(* CODESYS project MC516.project
   CompiledLibraryCompatibilityVersion: LeadSysStudio V3.5 SP15 Patch 4
   Title: MC516

Project tree, tasks and I/O mapping:
  Device : MC516, Leadshine Technology Co., Ltd., order no. 516101, version 3.5.15.40
      settings: RetainMode = 0; RetainStartAddr = 20480; RetainEndAddr = 524288; RetainSize = 524288
    application Application
      libraries: Standard, * (System)
      task EtherCAT_Master_Leadshine_A (cyclic, interval 2000 µs, priority 0) calls EtherCAT_Master_Leadshine_A.EtherCAT_Task, M
      program M [ST]: io, motion, save_check, save_apply, work
      DataMain/
        data type HMIData
        data type SaveData
      function block AxisFB [ST]: calculate_home_delta_μ, follow
      Enum/
        data type State
        data type JogType
      Object/
        data type Button
        data type Cylinder
        data type AxisEC
        data type AxisECFollow
        data type Problem
      function StateNext [ST]
      DataWork/
        data type SupplyData
        data type WorkData
        data type CutData
      function block CutFB [ST]
      visualisation Visualization
      function block SupplyFB [ST]
      Symbols
      global variables PersistentVars
      function block AxisFBSetTorqueLimit [ST]
      function block SimpleMotion [ST]
    Resource Usage
    Device Diagnose
    Network Configuration
      LocalBus Config
    SoftMotion General Axis Pool
      JogEncoder : SMC_FreeEncoder, 3S - Smart Software Solutions GmbH, order no. 1805, version 3.5.5.0
          settings: wDriveID = 3; dwRatioTechUnitsDenom = 400; ScalingIncs = 400
    High_Speed_IO_Module : High Speed IO, Leadshine Technology Co., Ltd., version 3.5.15.40
        settings: HS_IO_Mode_0.High In IO Mode 0 = 196611; HS_IO_Mode_0.High In IO Mode 2 = 196611; Counter_Mask = 5; Ioin_Mask = 19; HS counter 1.Counter_CountMode = 1; HS counter 2.Counter_CountMode = 1; HS counter 3.Counter_SetWorkMode = 2; HS counter 3.Counter_CountMode = 1; InputFilter Para.Time_In0 = 2; InputFilter Para.Time_In1 = 2; InputFilter Para.Time_In4 = 2
        unmapped channels: Genral_IO_IN, Genral_IO_Out
    LocalBus_Master_Module : LocalBus Master, Leadshine Technology Co., Ltd., version 3.5.15.40
    EtherCAT_Master_Leadshine_A : EtherCAT Master SoftMotion, 3S - Smart Software Solutions GmbH, version 3.5.16.30
        settings: MasterCycleTime = 2000; NetworkName = 'ecat'; SelectNetworkByName = TRUE; SrcAddress1 = 10; SrcAddress2 = 889192738
      XINJE_DS5C1_CoE_Drive_Rev4_0 : XINJE-DS5C1 EtherCAT(CoE) Drive Rev4.0 v3.7.70, Xinje Electronics, Inc., order no. XINJE-DS5C1 CoE Drive Rev4.0, version Revision=16#20201207
          settings: Number of Inputs = 6; Number of Infos about Inputs = 6; StationAlias = 1; Sync.Length = 17; FMMU.Length = 17; DC sync0 cycletime = 2000; DC sync1 cycletime = 2000; Number of SDO = 6; Interpolation time period.Value = 2; RxTxPdo.NumberofEntries = 6; RxTxPdo.Index = 16#1A00; RxTxPdo.DependOnSlot = False; RxTxPdo.DependOnSlotGroup = False; RxTxPdo.OverwrittenByModule = False; Status Word.Offset = 0; Status Word.DependOnSlot = False; Status Word.DependOnSlotGroup = False; ActualPosition.Offset = 0; ActualPosition.DependOnSlot = False; ActualPosition.DependOnSlotGroup = False; Velocity actual value.Offset = 0; Velocity actual value.DependOnSlot = False; Velocity actual value.DependOnSlotGroup = False; ActualTorque.Offset = 0; ActualTorque.DependOnSlot = False; ActualTorque.DependOnSlotGroup = False; ModeOfOperationDisplay.Offset = 0; ModeOfOperationDisplay.DependOnSlot = False; ModeOfOperationDisplay.DependOnSlotGroup = False; Index = 16#5000; SubIndex = 0; Size = 32; Offset = 0; DependOnSlot = False; DependOnSlotGroup = False; Status Word.Default = ''; Status Word.Comment = ''; ActualPosition.Default = ''; ActualPosition.Comment = ''; Velocity actual value.Default = '';
            Velocity actual value.Comment = ''; ActualTorque.Default = ''; ActualTorque.Comment = ''; ModeOfOperationDisplay.Default = ''; ModeOfOperationDisplay.Comment = ''; Name = 'Encode Single Position'; DataType = 'DINT'; Default = ''; Comment = ''
          unmapped channels: Control Word, TargetPosition, TargetVelocity, TargetTorque, ModeOfOperation, Status Word, ActualPosition, Velocity actual value, ActualTorque, ModeOfOperationDisplay, Encode Single Position
        Axis : Axis, 3S - Smart Software Solutions GmbH, order no. 0, version 4.6.1.0
            settings: wDriveID = 0; dwRatioTechUnitsDenom = 1; eRampType = 3; Number of pulses for one revolution = 131072; The displacement for one revolution of the workbench = 131072; Gear ratio molecule = 1; Gear ratio denominator = 1; ScalingIncs = 131072; InvertDirection = False; AdrOffset_8010 = 4; BitOffset_8010 = 0; BitLength_8010 = 16; Address_8010 = '%QW2'; Type_8010 = 'UINT'; AddressPointer_8010 = ADR(%QW2); AdrOffset_8020 = 8; BitOffset_8020 = 0; BitLength_8020 = 32; Address_8020 = '%QD2'; Type_8020 = 'DINT'; AddressPointer_8020 = ADR(%QD2); AdrOffset_8030 = 12; BitOffset_8030 = 0; BitLength_8030 = 32; Address_8030 = '%QD3'; Type_8030 = 'DINT'; AddressPointer_8030 = ADR(%QD3); AdrOffset_8040 = 16; BitOffset_8040 = 0; BitLength_8040 = 16; Address_8040 = '%QW8'; Type_8040 = 'INT'; AddressPointer_8040 = ADR(%QW8); AdrOffset_8050 = 18; BitOffset_8050 = 0; BitLength_8050 = 8; Address_8050 = '%QB18'; Type_8050 = 'SINT'; AddressPointer_8050 = ADR(%QB18); AdrOffset_8060 = 4294967295;
              BitOffset_8060 = 0; BitLength_8060 = 0; Address_8060 = ''; Type_8060 = ''; AddressPointer_8060 = 0; AdrOffset_8070 = 4294967295; BitOffset_8070 = 0; BitLength_8070 = 0; Address_8070 = ''; Type_8070 = ''; AddressPointer_8070 = 0; AdrOffset_8080 = 4294967295; BitOffset_8080 = 0; BitLength_8080 = 0; Address_8080 = ''; Type_8080 = ''; AddressPointer_8080 = 0; AdrOffset_8090 = 4294967295; BitOffset_8090 = 0; BitLength_8090 = 0; Address_8090 = ''; Type_8090 = ''; AddressPointer_8090 = 0; AdrOffset_8510 = 4; BitOffset_8510 = 0; BitLength_8510 = 16; Address_8510 = '%IW2'; Type_8510 = 'UINT'; AddressPointer_8510 = ADR(%IW2); AdrOffset_8520 = 8; BitOffset_8520 = 0; BitLength_8520 = 32; Address_8520 = '%ID2'; Type_8520 = 'DINT'; AddressPointer_8520 = ADR(%ID2); AdrOffset_8530 = 12; BitOffset_8530 = 0; BitLength_8530 = 32; Address_8530 = '%ID3'; Type_8530 = 'DINT';
              AddressPointer_8530 = ADR(%ID3); AdrOffset_8540 = 16; BitOffset_8540 = 0; BitLength_8540 = 16; Address_8540 = '%IW8'; Type_8540 = 'INT'; AddressPointer_8540 = ADR(%IW8); AdrOffset_8550 = 18; BitOffset_8550 = 0; BitLength_8550 = 8; Address_8550 = '%IB18'; Type_8550 = 'SINT'; AddressPointer_8550 = ADR(%IB18); AdrOffset_8560 = 4294967295; BitOffset_8560 = 0; BitLength_8560 = 0; Address_8560 = ''; Type_8560 = ''; AddressPointer_8560 = 0; AdrOffset_8570 = 4294967295; BitOffset_8570 = 0; BitLength_8570 = 0; Address_8570 = ''; Type_8570 = ''; AddressPointer_8570 = 0; AdrOffset_8580 = 4294967295; BitOffset_8580 = 0; BitLength_8580 = 0; Address_8580 = ''; Type_8580 = ''; AddressPointer_8580 = 0; AdrOffset_8590 = 4294967295; BitOffset_8590 = 0; BitLength_8590 = 0; Address_8590 = ''; Type_8590 = ''; AddressPointer_8590 = 0; AdrOffset_8600 = 4294967295; BitOffset_8600 = 0; BitLength_8600 = 0;
              Address_8600 = ''; Type_8600 = ''; AddressPointer_8600 = 0; AdrOffset_8600 = 4294967295; BitOffset_8600 = 0; BitLength_8600 = 0; Address_8610 = ''; Type_8610 = ''; AddressPointer_8610 = 0; AdrOffset_8620 = 4294967295; BitOffset_8620 = 0; BitLength_8620 = 0; Address_8620 = ''; Type_8620 = ''; AddressPointer_8620 = 0
      XINJE_DS5C1_CoE_Drive_Rev4_0_1 : XINJE-DS5C1 EtherCAT(CoE) Drive Rev4.0 v3.7.70, Xinje Electronics, Inc., order no. XINJE-DS5C1 CoE Drive Rev4.0, version Revision=16#20201207
          settings: Number of Inputs = 6; Number of Infos about Inputs = 6; StationAlias = 1; Optional = False; DeviceIdenticationADO = 0; DeviceIdenticationMode = 0; Sync.Length = 17; FMMU.Length = 17; DC sync0 cycletime = 2000; DC sync1 cycletime = 2000; Number of SDO = 5; Interpolation time period.Value = 2; RxTxPdo.NumberofEntries = 6; RxTxPdo.Index = 16#1A00; RxTxPdo.DependOnSlot = False; RxTxPdo.DependOnSlotGroup = False; RxTxPdo.OverwrittenByModule = False; Status Word.Offset = 0; Status Word.DependOnSlot = False; Status Word.DependOnSlotGroup = False; ActualPosition.Offset = 0; ActualPosition.DependOnSlot = False; ActualPosition.DependOnSlotGroup = False; Velocity actual value.Offset = 0; Velocity actual value.DependOnSlot = False; Velocity actual value.DependOnSlotGroup = False; ActualTorque.Offset = 0; ActualTorque.DependOnSlot = False; ActualTorque.DependOnSlotGroup = False; ModeOfOperationDisplay.Offset = 0; ModeOfOperationDisplay.DependOnSlot = False; ModeOfOperationDisplay.DependOnSlotGroup = False; Index = 16#5000; SubIndex = 0; Size = 32; Offset = 0; DependOnSlot = False; DependOnSlotGroup = False; Status Word.Default = ''; Status Word.Comment = '';
            ActualPosition.Default = ''; ActualPosition.Comment = ''; Velocity actual value.Default = ''; Velocity actual value.Comment = ''; ActualTorque.Default = ''; ActualTorque.Comment = ''; ModeOfOperationDisplay.Default = ''; ModeOfOperationDisplay.Comment = ''; Name = 'Encode Single Position'; DataType = 'DINT'; Default = ''; Comment = ''
          unmapped channels: Control Word, TargetPosition, TargetVelocity, TargetTorque, ModeOfOperation, Status Word, ActualPosition, Velocity actual value, ActualTorque, ModeOfOperationDisplay, Encode Single Position
        Axis_1 : Axis, 3S - Smart Software Solutions GmbH, order no. 0, version 4.6.1.0
            settings: dwRatioTechUnitsDenom = 1; eRampType = 3; Number of pulses for one revolution = 131072; The displacement for one revolution of the workbench = 131072; Gear ratio molecule = 1; Gear ratio denominator = 1; ScalingIncs = 131072; InvertDirection = False; AdrOffset_8010 = 20; BitOffset_8010 = 0; BitLength_8010 = 16; Address_8010 = '%QW10'; Type_8010 = 'UINT'; AddressPointer_8010 = ADR(%QW10); AdrOffset_8020 = 24; BitOffset_8020 = 0; BitLength_8020 = 32; Address_8020 = '%QD6'; Type_8020 = 'DINT'; AddressPointer_8020 = ADR(%QD6); AdrOffset_8030 = 28; BitOffset_8030 = 0; BitLength_8030 = 32; Address_8030 = '%QD7'; Type_8030 = 'DINT'; AddressPointer_8030 = ADR(%QD7); AdrOffset_8040 = 32; BitOffset_8040 = 0; BitLength_8040 = 16; Address_8040 = '%QW16'; Type_8040 = 'INT'; AddressPointer_8040 = ADR(%QW16); AdrOffset_8050 = 34; BitOffset_8050 = 0; BitLength_8050 = 8; Address_8050 = '%QB34'; Type_8050 = 'SINT'; AddressPointer_8050 = ADR(%QB34); AdrOffset_8060 = 4294967295; BitOffset_8060 = 0;
              BitLength_8060 = 0; Address_8060 = ''; Type_8060 = ''; AddressPointer_8060 = 0; AdrOffset_8070 = 4294967295; BitOffset_8070 = 0; BitLength_8070 = 0; Address_8070 = ''; Type_8070 = ''; AddressPointer_8070 = 0; AdrOffset_8080 = 4294967295; BitOffset_8080 = 0; BitLength_8080 = 0; Address_8080 = ''; Type_8080 = ''; AddressPointer_8080 = 0; AdrOffset_8090 = 4294967295; BitOffset_8090 = 0; BitLength_8090 = 0; Address_8090 = ''; Type_8090 = ''; AddressPointer_8090 = 0; AdrOffset_8510 = 24; BitOffset_8510 = 0; BitLength_8510 = 16; Address_8510 = '%IW12'; Type_8510 = 'UINT'; AddressPointer_8510 = ADR(%IW12); AdrOffset_8520 = 28; BitOffset_8520 = 0; BitLength_8520 = 32; Address_8520 = '%ID7'; Type_8520 = 'DINT'; AddressPointer_8520 = ADR(%ID7); AdrOffset_8530 = 32; BitOffset_8530 = 0; BitLength_8530 = 32; Address_8530 = '%ID8'; Type_8530 = 'DINT'; AddressPointer_8530 = ADR(%ID8);
              AdrOffset_8540 = 36; BitOffset_8540 = 0; BitLength_8540 = 16; Address_8540 = '%IW18'; Type_8540 = 'INT'; AddressPointer_8540 = ADR(%IW18); AdrOffset_8550 = 38; BitOffset_8550 = 0; BitLength_8550 = 8; Address_8550 = '%IB38'; Type_8550 = 'SINT'; AddressPointer_8550 = ADR(%IB38); AdrOffset_8560 = 4294967295; BitOffset_8560 = 0; BitLength_8560 = 0; Address_8560 = ''; Type_8560 = ''; AddressPointer_8560 = 0; AdrOffset_8570 = 4294967295; BitOffset_8570 = 0; BitLength_8570 = 0; Address_8570 = ''; Type_8570 = ''; AddressPointer_8570 = 0; AdrOffset_8580 = 4294967295; BitOffset_8580 = 0; BitLength_8580 = 0; Address_8580 = ''; Type_8580 = ''; AddressPointer_8580 = 0; AdrOffset_8590 = 4294967295; BitOffset_8590 = 0; BitLength_8590 = 0; Address_8590 = ''; Type_8590 = ''; AddressPointer_8590 = 0; AdrOffset_8600 = 4294967295; BitOffset_8600 = 0; BitLength_8600 = 0; Address_8600 = '';
              Type_8600 = ''; AddressPointer_8600 = 0; AdrOffset_8600 = 4294967295; BitOffset_8600 = 0; BitLength_8600 = 0; Address_8610 = ''; Type_8610 = ''; AddressPointer_8610 = 0; AdrOffset_8620 = 4294967295; BitOffset_8620 = 0; BitLength_8620 = 0; Address_8620 = ''; Type_8620 = ''; AddressPointer_8620 = 0
      XINJE_DS5C1_CoE_Drive_Rev4_0_2 : XINJE-DS5C1 EtherCAT(CoE) Drive Rev4.0 v3.7.70, Xinje Electronics, Inc., order no. XINJE-DS5C1 CoE Drive Rev4.0, version Revision=16#20201207
          settings: Number of Inputs = 6; Number of Infos about Inputs = 6; StationAlias = 1; Optional = False; DeviceIdenticationADO = 0; DeviceIdenticationMode = 0; Sync.Length = 17; FMMU.Length = 17; DC sync0 cycletime = 2000; DC sync1 cycletime = 2000; Number of SDO = 8; Interpolation time period.Value = 2; RxTxPdo.NumberofEntries = 6; RxTxPdo.Index = 16#1A00; RxTxPdo.DependOnSlot = False; RxTxPdo.DependOnSlotGroup = False; RxTxPdo.OverwrittenByModule = False; Status Word.Offset = 0; Status Word.DependOnSlot = False; Status Word.DependOnSlotGroup = False; ActualPosition.Offset = 0; ActualPosition.DependOnSlot = False; ActualPosition.DependOnSlotGroup = False; Velocity actual value.Offset = 0; Velocity actual value.DependOnSlot = False; Velocity actual value.DependOnSlotGroup = False; ActualTorque.Offset = 0; ActualTorque.DependOnSlot = False; ActualTorque.DependOnSlotGroup = False; ModeOfOperationDisplay.Offset = 0; ModeOfOperationDisplay.DependOnSlot = False; ModeOfOperationDisplay.DependOnSlotGroup = False; Index = 16#5000; SubIndex = 0; Size = 32; Offset = 0; DependOnSlot = False; DependOnSlotGroup = False; Status Word.Default = ''; Status Word.Comment = '';
            ActualPosition.Default = ''; ActualPosition.Comment = ''; Velocity actual value.Default = ''; Velocity actual value.Comment = ''; ActualTorque.Default = ''; ActualTorque.Comment = ''; ModeOfOperationDisplay.Default = ''; ModeOfOperationDisplay.Comment = ''; Name = 'Encode Single Position'; DataType = 'DINT'; Default = ''; Comment = ''
          unmapped channels: Control Word, TargetPosition, TargetVelocity, TargetTorque, ModeOfOperation, Status Word, ActualPosition, Velocity actual value, ActualTorque, ModeOfOperationDisplay, Encode Single Position
        Axis_2 : Axis, 3S - Smart Software Solutions GmbH, order no. 0, version 4.6.1.0
            settings: wDriveID = 2; dwRatioTechUnitsDenom = 1; iMovementType = 0; fPositionPeriod = 360000; eRampType = 3; Number of pulses for one revolution = 131072; The displacement for one revolution of the workbench = 131072; Gear ratio molecule = 1; Gear ratio denominator = 1; ScalingIncs = 131072; InvertDirection = False; AdrOffset_8010 = 36; BitOffset_8010 = 0; BitLength_8010 = 16; Address_8010 = '%QW18'; Type_8010 = 'UINT'; AddressPointer_8010 = ADR(%QW18); AdrOffset_8020 = 40; BitOffset_8020 = 0; BitLength_8020 = 32; Address_8020 = '%QD10'; Type_8020 = 'DINT'; AddressPointer_8020 = ADR(%QD10); AdrOffset_8030 = 44; BitOffset_8030 = 0; BitLength_8030 = 32; Address_8030 = '%QD11'; Type_8030 = 'DINT'; AddressPointer_8030 = ADR(%QD11); AdrOffset_8040 = 48; BitOffset_8040 = 0; BitLength_8040 = 16; Address_8040 = '%QW24'; Type_8040 = 'INT'; AddressPointer_8040 = ADR(%QW24); AdrOffset_8050 = 50; BitOffset_8050 = 0; BitLength_8050 = 8; Address_8050 = '%QB50'; Type_8050 = 'SINT';
              AddressPointer_8050 = ADR(%QB50); AdrOffset_8060 = 4294967295; BitOffset_8060 = 0; BitLength_8060 = 0; Address_8060 = ''; Type_8060 = ''; AddressPointer_8060 = 0; AdrOffset_8070 = 4294967295; BitOffset_8070 = 0; BitLength_8070 = 0; Address_8070 = ''; Type_8070 = ''; AddressPointer_8070 = 0; AdrOffset_8080 = 4294967295; BitOffset_8080 = 0; BitLength_8080 = 0; Address_8080 = ''; Type_8080 = ''; AddressPointer_8080 = 0; AdrOffset_8090 = 4294967295; BitOffset_8090 = 0; BitLength_8090 = 0; Address_8090 = ''; Type_8090 = ''; AddressPointer_8090 = 0; AdrOffset_8510 = 44; BitOffset_8510 = 0; BitLength_8510 = 16; Address_8510 = '%IW22'; Type_8510 = 'UINT'; AddressPointer_8510 = ADR(%IW22); AdrOffset_8520 = 48; BitOffset_8520 = 0; BitLength_8520 = 32; Address_8520 = '%ID12'; Type_8520 = 'DINT'; AddressPointer_8520 = ADR(%ID12); AdrOffset_8530 = 52; BitOffset_8530 = 0; BitLength_8530 = 32;
              Address_8530 = '%ID13'; Type_8530 = 'DINT'; AddressPointer_8530 = ADR(%ID13); AdrOffset_8540 = 56; BitOffset_8540 = 0; BitLength_8540 = 16; Address_8540 = '%IW28'; Type_8540 = 'INT'; AddressPointer_8540 = ADR(%IW28); AdrOffset_8550 = 58; BitOffset_8550 = 0; BitLength_8550 = 8; Address_8550 = '%IB58'; Type_8550 = 'SINT'; AddressPointer_8550 = ADR(%IB58); AdrOffset_8560 = 4294967295; BitOffset_8560 = 0; BitLength_8560 = 0; Address_8560 = ''; Type_8560 = ''; AddressPointer_8560 = 0; AdrOffset_8570 = 4294967295; BitOffset_8570 = 0; BitLength_8570 = 0; Address_8570 = ''; Type_8570 = ''; AddressPointer_8570 = 0; AdrOffset_8580 = 4294967295; BitOffset_8580 = 0; BitLength_8580 = 0; Address_8580 = ''; Type_8580 = ''; AddressPointer_8580 = 0; AdrOffset_8590 = 4294967295; BitOffset_8590 = 0; BitLength_8590 = 0; Address_8590 = ''; Type_8590 = ''; AddressPointer_8590 = 0; AdrOffset_8600 = 4294967295;
              BitOffset_8600 = 0; BitLength_8600 = 0; Address_8600 = ''; Type_8600 = ''; AddressPointer_8600 = 0; AdrOffset_8600 = 4294967295; BitOffset_8600 = 0; BitLength_8600 = 0; Address_8610 = ''; Type_8610 = ''; AddressPointer_8610 = 0; AdrOffset_8620 = 4294967295; BitOffset_8620 = 0; BitLength_8620 = 0; Address_8620 = ''; Type_8620 = ''; AddressPointer_8620 = 0
  text list GlobalTextList
*)

// Device/Application/DataMain/HMIData
{ attribute 'pack_mode' := ''}
TYPE HMIData :
STRUCT
	//
	sv: SaveData;
	sv_trigger: BOOL;
	sv_need_check: BOOL;
	sv_need: BOOL;
	//
	plc_ready: BOOL;
	hmi_ready: BOOL;
	run: BOOL;
	stop: BOOL;
	home: BOOL;
	problem_fix: ARRAY[0..7] OF BOOL;
	//
	supply_test: BOOL;
	supply_arm_clamp_holder: BOOL;
	supply_arm_clamp: BOOL;
	supply_spindle_clamp: BOOL;
	supply_spindle_extract: BOOL;
	cut_spindle_run: BOOL;
	hydraulic_run: BOOL;
	jog_micro_per_sec_or_rev: UINT;
	//
	view_input: ARRAY[0..15] OF BOOL;
	view_input_jog_index: UINT;
	view_input_jog_micro: DINT;
	view_output: ARRAY[0..15] OF BOOL;
	//
	view_can_run: BOOL;
	view_can_stop: BOOL;
	view_can_home: BOOL;
	view_auto: BOOL;
	view_manual: BOOL;
	//
	view_axis_encoder: ARRAY[0..2] OF DINT;
	view_axis_micro: ARRAY[0..2] OF UDINT;
	view_axis_mNm: ARRAY[0..2] OF UDINT;
	view_cut_spindle_run_ing: BOOL;
	view_cut_spindle_rpm: UDINT;
	//
	view_supply_test: ARRAY[0..4] OF BOOL;
	//
	view_problem: ARRAY[0..7] OF BOOL;
	view_cycle_count: UDINT;
	view_cycle_time_msec: UDINT;
	//
	view_state: ARRAY[0..7] OF INT;
END_STRUCT
END_TYPE

// Device/Application/DataMain/SaveData
{ attribute 'pack_mode' := ''}
TYPE SaveData :
STRUCT
	set_done: BOOL;
	////////
	//SAME//
	////////
	cylinder_n_delay_msec: ARRAY[0..3] OF UINT;
	cylinder_p_delay_msec: ARRAY[0..3] OF UINT;
	//
	// (a) increments        <> (d) motor turns
	// (b) motor turns       <> (e) gear output turns
	// (c) gear output turns <> (f) units in application
	// .iRatioTechUnitsNum = gear_num = gear_dir * d * e * f 
	// .dwRatioTechUnitsDenom = gear_den = a * b * c
	max_rpm: ARRAY[0..2] OF UINT;
	gear_num: ARRAY[0..2] OF DINT;
	gear_den: ARRAY[0..2] OF DINT;
	gear_dir: ARRAY[0..2] OF BOOL;
	home_torque_mNm: ARRAY[0..2] OF UINT;
	home_encoder_value_recorded: BOOL;
	home_encoder_value: ARRAY[0..2] OF DINT;
	max_micro_recorded: BOOL;
	max_micro: ARRAY[0..2] OF DINT;
	overload_hold_torque_factor: ARRAY[0..2] OF UINT;
	overload_hold_torque_time_msec: ARRAY[0..2] OF UINT;
	overload_instant_torque_factor: ARRAY[0..2] OF UINT;
	ramp_time_msec: ARRAY[0..2] OF UINT;
	jerk_factor: ARRAY[0..2] OF UINT;
	///////////
	//MACHINE//
	///////////
	cut_begin_micro: ARRAY[0..1] OF DINT;
	cut_rapid_micro: ARRAY[0..1] OF DINT;
	cut_end_micro: ARRAY[0..1] OF DINT;
	cut_offset_micro: ARRAY[0..1] OF DINT;
	cut_lag_micro: UDINT;
	cut_rapid_micro_per_rev: UDINT;
	cut_micro_per_rev: UDINT;
	cut_dwell_msec: UINT;
	cut_retract_micro: UDINT; // vị trí lùi về
	cut_retract_micro_per_sec: UDINT; // tốc độ lùi sau khi cắt
	cut_spindle_encoder_resolution: UINT;
	//
	supply_begin_micro: DINT;
	supply_mid_micro: DINT;
	supply_end_micro: DINT;
	supply_micro_per_sec: DINT;
END_STRUCT
END_TYPE

// Device/Application/Enum/State
{attribute 'qualified_only'}
{attribute 'strict'}
TYPE State :
(
	NONE := 0,
	RST := 1,
	RST_DONE := 50,
	HOME := 51,
	HOME_FORWARD := 71,
	HOME_DONE := 90,
	HOME_OFFSET := 91,
	HOME_OFFSET_DONE := 99,
	READY := 100,
	RUN := 101,
	RUN_ING := 200
);
END_TYPE

// Device/Application/Object/Button
{ attribute 'pack_mode' := ''}
TYPE Button :
STRUCT
	on: BOOL;
	rise: R_TRIG;
	rise_physical: R_TRIG;
	fall: F_TRIG;
	fall_physical: F_TRIG;
	timer: TON;
END_STRUCT
END_TYPE

// Device/Application/Object/Cylinder
{ attribute 'pack_mode' := ''}
TYPE Cylinder :
STRUCT
	on: BOOL;
	n_timer: TON;
	p_timer: TON;
END_STRUCT
END_TYPE

// Device/Application/Object/AxisEC
{ attribute 'pack_mode' := ''}
TYPE AxisEC :
STRUCT
	///////
	//REF//
	///////
	ref: POINTER TO SM3_Drive_ETC_DS402_CyclicSync.AXIS_REF_ETC_DS402_CS;
	read: POINTER TO SMC3_ETC_ReadParameter_CoE;
	write: POINTER TO SMC3_ETC_WriteParameter_CoE;
	read_status: POINTER TO MC_ReadStatus;
	set_mode: POINTER TO SMC_SetControllerMode;
	power: POINTER TO MC_Power;
	reset: POINTER TO MC_Reset;
	stop: POINTER TO MC_Stop;
	inch: POINTER TO SMC_Inch;
	fsv: POINTER TO SMC_FollowSetValues;
	sp: POINTER TO MC_SetPosition;
	mabs: POINTER TO MC_MoveAbsolute;
	set_torque_limit: AxisFBSetTorqueLimit;
	////////
	//DATA//
	////////
	encoder_resolution: DINT;
	torque_rated_Nm: LREAL;
	encoder_single_position: DINT;
	///////////
	//PROCESS//
	///////////
	state: INT;
	torque_Nm: LREAL;
	torque_Nm_abs: LREAL;
	overload: BOOL;
	overload_check: BOOL;
	overload_hold_torque_Nm: LREAL;
	overload_hold_torque_timer: TON;
	overload_instant_torque_Nm: LREAL;
	//home
	home_done: BOOL; // = TRUE khi về gốc thành công, chỉ về gốc khi bật máy
	home_done_forward_ignore: BOOL;
	home_to_encoder: BOOL; //
	home_torque_Nm: LREAL;
	home_hit_timer: TON;
	home_hit_test: BOOL;
	home_offset_absolute_μ: LREAL; // vị trí từ điểm va chạm đến gốc tuyệt đối, xem hàm save_apply()
	home_back_μ_per_sec: LREAL; // tốc độ lùi về lấy gốc
	home_forward_μ_per_sec: LREAL; // tốc độ tiến sau khi lấy gốc xong
	home_offset_μ: LREAL; // giá trị này để thực hiện lệnh state = State.HOME_OFFSET ở trong AxisLinearFB
	home_encoder_value_recorded: BOOL;
	home_encoder_value_save: POINTER TO DINT; // pointer tới giá trị ở save data
	home_encoder_delta: DINT;
	home_delta_μ: LREAL;
	//
	ramp_time_sec: LREAL;
	jerk_factor: LREAL;
	//
	jog_type: JogType;
	jog_delta: LREAL;
	jog_velocity: LREAL;
	jog_acceleration: LREAL;
	max_μ_recorded: BOOL;
	max_μ_save: POINTER TO DINT;
	max_μ: LREAL; // giới hạn vị trí tối đa có thể di chuyển từ gốc tuyệt đối
	max_μ_per_sec: LREAL; // giới hạn tốc độ tối đa
	//run
	target_position_μ: LREAL; // sử dụng cho state = State.RUN ở trong AxisLinearFB
	target_velocity_μ_per_sec: LREAL; // sử dụng cho state = State.RUN ở trong AxisLinearFB
END_STRUCT
END_TYPE

// Device/Application/DataWork/SupplyData
{ attribute 'pack_mode' := ''}
TYPE SupplyData :
STRUCT
	state: INT;
	axis: AxisEC;
	axis_fb: AxisFB;
	state_ready: BOOL;
	//
	input_air: BOOL;
	input_hydraulic: BOOL;
	input_arm_clamp_holder_p: BOOL;
	input_feeder_small: BOOL;
	input_feeder_big: BOOL;
	hydraulic: BOOL;
	arm_clamp_holder: Cylinder;
	arm_clamp_holder_p_rise: R_TRIG;
	arm_clamp: Cylinder;
	spindle_clamp: Cylinder;
	spindle_clamp_release: BOOL;
	spindle_extract: Cylinder;
	//
	begin_μdeg: LREAL;
	mid_μdeg: LREAL;
	end_μdeg: LREAL;
	μdeg_per_sec: LREAL;
	foil_stuck: Problem;
END_STRUCT
END_TYPE

// Device/Application/DataWork/WorkData
{ attribute 'pack_mode' := ''}
TYPE WorkData :
STRUCT
	state: INT;
	//
	input_run: Button;
	input_stop: Button;
	input_home: Button;
	input_jog_index: UINT;
	//
	can_run: BOOL;
	can_stop: BOOL;
	can_home: BOOL;
	jog_i: POINTER TO AxisEC;
	jog_encoder_counter: LS_Counter;
	jog_encoder_counter_set: LS_PresetValue;
	jog_encoder: POINTER TO SM3_Basic.FREE_ENCODER_REF;
	jog_encoder_last: LREAL;
	run_auto: Button;
	overload: Problem;
	alarm: BOOL;
	//
	cut_spindle_run_rise: R_TRIG;
	cut_spindle_run_timer: TON;
	supply_hydraulic_rise: R_TRIG;
	supply_hydraulic_timer: TON;
	supply_test_timer: TON;
	//
	manual_active: BOOL;
	final_cycle_flag: BOOL;
	final_cycle: BOOL;
	cycle_start_msec: ULINT;
	cycle_time_msec: UDINT;
END_STRUCT
END_TYPE

// Device/Application/DataWork/CutData
{ attribute 'pack_mode' := ''}
TYPE CutData :
STRUCT
	state: INT;
	axiss: ARRAY[0..1] OF AxisEC;
	axiss_fb: ARRAY[0..1] OF AxisFB;
	//
	state_spindle: INT;
	spindle: BOOL;
	spindle_encoder_counter_last: DINT;
	spindle_encoder_counter: LS_Counter;
	spindle_encoder_resolution: UDINT;
	spindle_encoder_time_msec_last: ULINT;
	spindle_rps_last: LREAL;
	spindle_rps: LREAL;
	spindle_rps_stable_cycle: INT;
	time_msec: ULINT;
	time_delta_sec: LREAL;
	//
	begin_μm: ARRAY[0..1] OF LREAL;
	rapid_μm: ARRAY[0..1] OF LREAL;
	end_μm: ARRAY[0..1] OF LREAL;
	lag_μm: LREAL;
	rapid_μm_per_rev: LREAL;
	μm_per_rev: LREAL;
	dwell_timer: TON;
	retract_μm: LREAL;
	retract_μm_per_sec: LREAL;
END_STRUCT
END_TYPE

// Device/Application/Enum/JogType
{attribute 'qualified_only'}
{attribute 'strict'}
TYPE JogType :
(
	NONE := 0,
	INCH := 1, // inch function
	FSV := 2 // follow set value function
);
END_TYPE

// Device/Application/Object/AxisECFollow
TYPE AxisECFollow :
STRUCT
	target: POINTER TO SM3_Basic.AXIS_REF_SM3;
	ratio: LREAL;
	offset: LREAL;
	offset_motion: SimpleMotion;
	//
	self_begin: LREAL;
	target_begin: LREAL;
	target_delta: LREAL;
	//
	deviation: LREAL;
END_STRUCT
END_TYPE

// Device/Application/Object/Problem
TYPE Problem :
STRUCT
	on: BOOL;
	timer: TON;
	rise: R_TRIG;
	fix_rise: R_TRIG;
	fix_timer: TON;
END_STRUCT
END_TYPE

// Device/Application/PersistentVars
{attribute 'qualified_only'}
VAR_GLOBAL PERSISTENT RETAIN
END_VAR
VAR_GLOBAL PERSISTENT
	M.save: SaveData;
END_VAR

// Device/Application/M
PROGRAM M
VAR
	time_msec_last: ULINT;
	time_msec : ULINT;
	time_delta_sec: LREAL;
	//
	axiss: ARRAY [0..2] OF POINTER TO SM3_Drive_ETC_DS402_CyclicSync.AXIS_REF_ETC_DS402_CS;
	// dùng pointer để dễ dàng thao tác với nhiều trục hơn, xem hàm motion()
	axiss_read: ARRAY[0..2] OF SMC3_ETC_ReadParameter_CoE;
	axiss_write: ARRAY[0..2] OF SMC3_ETC_WriteParameter_CoE;
	axiss_read_status: ARRAY[0..2] OF MC_ReadStatus;
	axiss_change_gearing_ratio: ARRAY[0..2] OF SMC_ChangeGearingRatio;
	axiss_reinit_drive: ARRAY[0..2] OF SMC3_ReinitDrive;
	axiss_set_mode: ARRAY[0..2] OF SMC_SetControllerMode;
	axiss_power: ARRAY[0..2] OF MC_Power; // bật tắt động cơ
	axiss_reset: ARRAY[0..2] OF MC_Reset; // reset lỗi
	axiss_stop: ARRAY[0..2] OF MC_Stop; // dừng
	axiss_inch: ARRAY[0..2] OF SMC_Inch;
	axiss_fsv: ARRAY[0..2] OF SMC_FollowSetValues;
	axiss_sp: ARRAY[0..2] OF MC_SetPosition;
	axiss_mabs: ARRAY[0..2] OF MC_MoveAbsolute;
	axiss_encoder_resolution: ARRAY[0..2] OF DINT;
	axiss_rated_torque_Nm: ARRAY[0..2] OF LREAL;
	axiss_max_rpm: ARRAY[0..2] OF UINT;
	axiss_max_μ_per_sec: ARRAY[0..2] OF LREAL;
	axiss_ready_all: BOOL;
	//
	state_main: INT;
	motion_active: BOOL;
	main_save: Button;
	supply_data: SupplyData;
	supply_fb: SupplyFB;
	cut_data: CutData;
	cut_fb: CutFB;
	work_data: WorkData;
	hmi: HMIData;
	//
	i: INT;
	j: INT;
	k: INT;
	axis_ec_i: POINTER TO AxisEC;
	axis_fb_i: POINTER TO AxisFB;
	cylinder_i: POINTER TO Cylinder;
	//
	test: BOOL;
END_VAR

VAR CONSTANT
	c_axis_i_max: INT := 4 - 1;
	c_cylinder_i_max: INT := 4 - 1;
	c_air_burst_i_max: INT := 2 - 1;
END_VAR

VAR RETAIN
	cycle_count: UDINT;
	cycle_count_reset_time_msec: ULINT;
END_VAR

VAR PERSISTENT
	save: SaveData;
END_VAR

MC_SysLib.SysTimeRtc.SysTimeRtcHighResGet(pTimestamp:= time_msec);
time_delta_sec := ULINT_TO_LREAL(time_msec - time_msec_last) * 1E-3;
time_msec_last := time_msec;
hmi.view_state[0] := state_main;
IF motion_active THEN
	motion();
END_IF
CASE state_main OF
	State.NONE: // khi khởi động thì state_main = 0 tức là = State.NONE
		test := FALSE;
		axiss[0] := ADR(Axis); // k = ADR(x) viết tắt cho "address of x" là hàm để lấy giá trị con trỏ (pointer) về biến x
		axiss[1] := ADR(Axis_1); // ví dụ muốn thay đổi giá trị của x ta sẽ viết k^ = 12345
		axiss[2] := ADR(Axis_2);
		axiss_change_gearing_ratio[0].iMovementType := SMC_MOVEMENTTYPE.linear;
		axiss_change_gearing_ratio[1].iMovementType := SMC_MOVEMENTTYPE.linear;
		axiss_change_gearing_ratio[2].iMovementType := SMC_MOVEMENTTYPE.linear;
		axiss_change_gearing_ratio[0].fPositionPeriod := 1_000;
		axiss_change_gearing_ratio[1].fPositionPeriod := 1_000;
		axiss_change_gearing_ratio[2].fPositionPeriod := 1_000;
		work_data.jog_encoder := ADR(JogEncoder);
		motion_active := FALSE;
		test := FALSE;
		StateNext(state_main); // chuyển tới trạng thái tiếp theo
	1:
		FOR i := 0 TO c_axis_i_max BY 1 DO // hàm FOR, FOR i = 0 TO 3 BY 1 DO sẽ chạy 4 lần i = [0, 1, 2, 3]
			CASE i OF // hàm CASE, lựa chọn theo giá trị i
				0:
					axis_ec_i := ADR(cut_data.axiss[0]);
					axis_fb_i := ADR(cut_data.axiss_fb[0]);
				1:
					axis_ec_i := ADR(cut_data.axiss[1]);
					axis_fb_i := ADR(cut_data.axiss_fb[1]);
				2:
					axis_ec_i := ADR(supply_data.axis);
					axis_fb_i := ADR(supply_data.axis_fb);
			END_CASE
			axis_ec_i^.ref := axiss[i];
			axis_ec_i^.read := ADR(axiss_read[i]);
			axis_ec_i^.write := ADR(axiss_write[i]);
			axis_ec_i^.read_status := ADR(axiss_read_status[i]);
			axis_ec_i^.set_mode := ADR(axiss_set_mode[i]);
			axis_ec_i^.power := ADR(axiss_power[i]);
			axis_ec_i^.reset := ADR(axiss_reset[i]);
			axis_ec_i^.stop := ADR(axiss_stop[i]);
			axis_ec_i^.inch := ADR(axiss_inch[i]);
			axis_ec_i^.fsv := ADR(axiss_fsv[i]);
			axis_ec_i^.sp := ADR(axiss_sp[i]);
			axis_ec_i^.mabs := ADR(axiss_mabs[i]);
			axis_fb_i^.d := axis_ec_i;
		END_FOR
		StateNext(state_main);
	2:
		axiss_ready_all := TRUE; // biến tạm thời để kiểm tra tất cả các servo đã hoàn thành lệnh hay chưa
		FOR i := 0 TO c_axis_i_max BY 1 DO
			axiss_ready_all := axiss_ready_all AND axiss[i]^.wCommunicationState = 100;
		END_FOR
		IF axiss_ready_all THEN // hoàn thành kết nối tất cả servo, ta đên bước tiếp theo
			motion_active := TRUE;
			state_main := 11;
		END_IF
	11: // đọc số xung encoder của servo
		FOR i := 0 TO c_axis_i_max BY 1 DO
			axiss_read[i].uiIndex := 16#608F; // mở ETHERCAT/XINJE_DS5C1.../ xem trong mục "CoE Online"
			axiss_read[i].usiSubIndex := 1; //
			axiss_read[i].xExecute := TRUE;
		END_FOR
		StateNext(state_main);
	12:
		axiss_ready_all := TRUE;
		FOR i := 0 TO c_axis_i_max BY 1 DO
			axiss_ready_all := axiss_ready_all AND axiss_read[i].xDone;
		END_FOR
		IF axiss_ready_all THEN
			FOR i := 0 TO c_axis_i_max BY 1 DO
				axiss_read[i].xExecute := FALSE;
				// Sau thực hiện hàm thành công phải đặt Execute = FALSE để cho lần đọc tiếp theo
				// vì đa số hàm chỉ chạy khi Execute chuyển từ FALSE sang TRUE (Rising edge)
				// xem Defination của hàm đê biết thêm chi tiết
				axiss_encoder_resolution[i] := DWORD_TO_DINT(axiss_read[i].dwValue);
			END_FOR
			StateNext(state_main);
		END_IF
	13: // đọc momen max của servo
		FOR i := 0 TO c_axis_i_max BY 1 DO
			axiss_read[i].uiIndex := 16#6076;
			axiss_read[i].usiSubIndex := 0;
			axiss_read[i].xExecute := TRUE;
		END_FOR
		StateNext(state_main);
	14:
		axiss_ready_all := TRUE;
		FOR i := 0 TO c_axis_i_max BY 1 DO
			axiss_ready_all := axiss_ready_all AND axiss_read[i].xDone;
		END_FOR
		IF axiss_ready_all THEN
			FOR i := 0 TO c_axis_i_max BY 1 DO
				axiss_read[i].xExecute := FALSE;
				axiss_rated_torque_Nm[i] := DWORD_TO_LREAL(axiss_read[i].dwValue) * 1E-3;
			END_FOR
			StateNext(state_main);
		END_IF
	15: // đọc max rpm của servo
		FOR i := 0 TO c_axis_i_max BY 1 DO
			axiss_read[i].uiIndex := 16#6080;
			axiss_read[i].usiSubIndex := 0;
			axiss_read[i].xExecute := TRUE;
		END_FOR
		StateNext(state_main);
	16:
		axiss_ready_all := TRUE;
		FOR i := 0 TO c_axis_i_max BY 1 DO
			axiss_ready_all := axiss_ready_all AND axiss_read[i].xDone;
		END_FOR
		IF axiss_ready_all THEN
			FOR i := 0 TO c_axis_i_max BY 1 DO
				axiss_read[i].xExecute := FALSE;
				axiss_max_rpm[i] := DWORD_TO_UINT(axiss_read[i].dwValue);
			END_FOR
			StateNext(state_main);
		END_IF
	17:
		FOR i := 0 TO c_axis_i_max BY 1 DO
			CASE i OF
				0: axis_ec_i := ADR(cut_data.axiss[0]);
				1: axis_ec_i := ADR(cut_data.axiss[1]);
				2: axis_ec_i := ADR(supply_data.axis);
			END_CASE
			axis_ec_i^.encoder_resolution := axiss_encoder_resolution[i];
			axis_ec_i^.torque_rated_Nm := axiss_rated_torque_Nm[i];
		END_FOR
		IF NOT save.set_done THEN
			save.set_done := TRUE;
			// biến "set_done" này nằm trong cấu trúc "save_data" nhằm mục đích
			// gán giá trị đầu cho biến lưu, đảm bảo đoạn gán dữ liệu này chỉ chạy 1 lần khi
			// PLC chạy lần dầu sau khi nạp lại chương trình.
			FOR i := 0 TO c_cylinder_i_max DO
				save.cylinder_n_delay_msec[i] := 0_200 + INT_TO_UINT(i * 2);
				save.cylinder_p_delay_msec[i] := 0_200 + INT_TO_UINT(i * 2 + 1);
			END_FOR
			//
			save.home_encoder_value_recorded := FALSE;
			save.max_micro_recorded := TRUE;
			FOR i := 0 TO c_axis_i_max BY 1 DO
				save.max_rpm[i] := 3000;
				save.gear_dir[i] := TRUE;
				save.gear_num[i] := axiss_encoder_resolution[i] / 2;
				save.gear_den[i] := axiss_encoder_resolution[i];
				save.home_torque_mNm[i] := 0_797; // 100 kg of force with 5mm ball screw
				save.home_encoder_value[i] := 0;
				save.max_micro[i] := 80_000;
				save.overload_hold_torque_factor[i] := 0_900 + INT_TO_UINT(i);
				save.overload_hold_torque_time_msec[i] := 1_000 + INT_TO_UINT(i);
				save.overload_instant_torque_factor[i] := 2_900 + INT_TO_UINT(i);
				save.ramp_time_msec[i] := 0_100;
				save.jerk_factor[i] := 30;
			END_FOR
			//
			save.cut_begin_micro[0] := 46_000;
			save.cut_begin_micro[1] := 46_000;
			save.cut_rapid_micro[0] := 51_000;
			save.cut_rapid_micro[1] := 51_000;
			save.cut_end_micro[0] := 53_500;
			save.cut_end_micro[1] := 53_500;
			save.cut_offset_micro[0] := -9_000;
			save.cut_offset_micro[1] := -9_000;
			//
			save.cut_lag_micro := 0_500;
			save.cut_rapid_micro_per_rev := 0_300; // => 0.4 * 50 = 20_000 μm/s
			save.cut_micro_per_rev := 0_025; // spindle 3000 rpm = 50 rps => cut_micron_per_sec = 0_2 * 50 = 10_000 μm/s
			save.cut_dwell_msec := 0_020;
			save.cut_retract_micro := 30_000;
			save.cut_retract_micro_per_sec := 150_000;
			save.cut_spindle_encoder_resolution := 1;
			//
			save.supply_begin_micro := 10_000;
			save.supply_mid_micro := 90_000;
			save.supply_end_micro := 100_000;
			save.supply_micro_per_sec := 180_000;
		END_IF
		StateNext(state_main);
	18:// set gear
		FOR i := 0 TO c_axis_i_max BY 1 DO
			axiss_change_gearing_ratio[i].iRatioTechUnitsNum := (BOOL_TO_DINT(save.gear_dir[i]) * 2 - 1) * save.gear_num[i];
			axiss_change_gearing_ratio[i].dwRatioTechUnitsDenom := DINT_TO_DWORD(save.gear_den[i]);
			axiss_change_gearing_ratio[i].bExecute := TRUE;
		END_FOR
		StateNext(state_main);
	19:// set gear done
		axiss_ready_all := TRUE;
		FOR i := 0 TO c_axis_i_max BY 1 DO
			axiss_ready_all := axiss_ready_all AND axiss_change_gearing_ratio[i].bDone AND NOT axiss_change_gearing_ratio[i].bError;
		END_FOR
		IF axiss_ready_all THEN
			FOR i := 0 TO c_axis_i_max BY 1 DO
				axiss_change_gearing_ratio[i].bExecute := FALSE;
			END_FOR
			StateNext(state_main);
		END_IF
	20:// reinit drive
		FOR i := 0 TO c_axis_i_max BY 1 DO
			axiss_reinit_drive[i].bExecute := TRUE;
		END_FOR
		StateNext(state_main);
	21:// reinit drive done
		axiss_ready_all := TRUE;
		FOR i := 0 TO c_axis_i_max BY 1 DO
			axiss_ready_all := axiss_ready_all AND axiss_reinit_drive[i].bDone AND axiss[i]^.wCommunicationState = 100;
		END_FOR
		IF axiss_ready_all THEN
			FOR i := 0 TO c_axis_i_max BY 1 DO
				axiss_reinit_drive[i].bExecute := FALSE;
			END_FOR
			StateNext(state_main);
		END_IF
	22:// calculate max
		FOR i := 0 TO c_axis_i_max BY 1 DO
			axiss_max_μ_per_sec[i] := (axiss_encoder_resolution[i] * (MIN(axiss_max_rpm[i], save.max_rpm[i]) / 60)) / ABS(axiss[i]^.fScalefactor);
		END_FOR
		StateNext(state_main);
	23:// prepair
		FOR i := 0 TO c_axis_i_max BY 1 DO
			axiss_power[i].Enable := TRUE;
			axiss_power[i].bRegulatorOn := TRUE;
		END_FOR
		StateNext(state_main);
	24:
		save_apply();
		StateNext(state_main);
	25:
		hmi.plc_ready := TRUE; // sau khi đã khởi động Servo bla bla thì ta PLC ready
		work_data.state := State.RST; // reset work
		state_main := State.RUN_ING; // bước vào giai đoạn chạy
		supply_fb.d := ADR(supply_data);
		cut_fb.d := ADR(cut_data);
	State.RUN_ING:
		io(); // kiểm tra io (gồm PLC io và HMI)
		supply_fb(d:= ); // hàm điều khiển cơ cấu cấp phôi (gồm servo và các xylanh khí nén)
		cut_fb(d:= ); // hàm điều khiển trục cắt
		work(); // hàm phối hợp giữa cấp phôi và cắt
END_CASE

ACTION io:
////////////
//HMI DOWN//
///////////
IF hmi.hmi_ready THEN
	////////
	//WORK//
	////////
	work_data.input_run.rise(CLK:= hmi.run, Q=> );
	work_data.input_stop.rise(CLK:= hmi.stop, Q=> );
	work_data.input_home.rise(CLK:= hmi.home, Q=> );
	work_data.overload.fix_rise(CLK:= hmi.problem_fix[0], Q=> );
	work_data.supply_hydraulic_rise(CLK:= hmi.hydraulic_run, Q=> );
	work_data.supply_hydraulic_timer(IN:= hmi.hydraulic_run, PT:= , Q=> , ET=> );
	work_data.supply_test_timer(IN:= hmi.supply_test, PT:= , Q=> , ET=> );
	work_data.cut_spindle_run_rise(CLK:= hmi.cut_spindle_run, Q=> );
	work_data.cut_spindle_run_timer(IN:= hmi.cut_spindle_run, PT:= , Q=> , ET=> );
	supply_data.foil_stuck.fix_rise(CLK:= hmi.problem_fix[1], Q=> );
	supply_data.foil_stuck.fix_timer(IN:= hmi.problem_fix[1], PT:= , Q=> , ET=> );
	////////
	//SAVE//
	////////
	IF hmi.sv_need_check THEN
		save_check();
		hmi.sv_need_check := FALSE;
	END_IF
	main_save.rise(CLK:= hmi.sv_trigger, Q=> ); // Trên HMI sẽ xuất hiện nút save khi biến hmi_data.save_need = true.
	IF main_save.rise.Q THEN
		save := hmi.sv;
		save_apply();
		hmi.sv_need := FALSE;
		hmi.sv_trigger := FALSE;
	END_IF
END_IF
/////////
//INPUT//
/////////
cut_data.axiss[0].encoder_single_position := DWORD_TO_DINT(%ID5);
cut_data.axiss[1].encoder_single_position := DWORD_TO_DINT(%ID10);
supply_data.axis.encoder_single_position := DWORD_TO_DINT(%ID15);
cut_data.time_msec := time_msec;
//
//jog encoder A phase %IX0.0
//jog encoder B phase %IX0.1
work_data.jog_encoder_counter(xEnable:= work_data.state = State.READY, eChannel:= COUNTER0, xValid=> , xError=> , eErrorID=> , diValue=> work_data.jog_encoder^.diEncoderPosition);
work_data.jog_encoder_counter_set(xExecute:= , eChannel:= COUNTER0, eTriggerEdge:= , diPresetValue:= , xDone=> , xBusy=> , xError=> , eErrorID=> );
work_data.input_run.rise_physical.CLK := %IX0.2;
work_data.input_stop.fall_physical.CLK := %IX0.3;
//spindle encoder %IX0.4
cut_data.spindle_encoder_counter(xEnable:= TRUE, eChannel:= COUNTER2, xValid=> , xError=> , eErrorID=> , diValue=> );
supply_data.input_feeder_small := %IX0.5;
supply_data.input_feeder_big := %IX0.6;
//empty %IX0.7
work_data.input_jog_index := (BOOL_TO_UINT(%IX1.0) +
										BOOL_TO_UINT(%IX1.1) * 2);
//empty %IX1.2 -> control panel
//empty %IX1.3 -> control panel
IF NOT test THEN
	supply_data.input_air := %IX1.4;
	supply_data.input_hydraulic := %IX1.5;
END_IF
supply_data.input_arm_clamp_holder_p := %IX1.6;
//empty %IX1.7
//
work_data.can_run := work_data.input_stop.fall_physical.CLK AND supply_data.input_air AND supply_data.input_hydraulic AND work_data.state = State.READY;
work_data.can_stop := work_data.state >= State.NONE;
work_data.can_home := work_data.state = State.RST_DONE OR work_data.state = State.READY;
IF cut_data.axiss[0].overload OR cut_data.axiss[1].overload OR supply_data.axis.overload THEN
	work_data.overload.on := TRUE;
END_IF
IF work_data.overload.fix_rise.Q THEN
	cut_data.axiss[0].overload := FALSE;
	cut_data.axiss[1].overload := FALSE;
	supply_data.axis.overload := FALSE;
	cut_data.axiss[0].overload_hold_torque_timer.IN := FALSE;
	cut_data.axiss[1].overload_hold_torque_timer.IN := FALSE;
	supply_data.axis.overload_hold_torque_timer.IN := FALSE;
	work_data.overload.on := FALSE;
END_IF
//
work_data.input_run.rise_physical(CLK:= , Q=> );
work_data.input_stop.fall_physical(CLK:= , Q=> );
work_data.input_run.timer(IN:= work_data.input_run.rise.CLK OR work_data.input_run.rise_physical.CLK, PT:= , Q=> , ET=> );
work_data.run_auto.timer(IN:= work_data.input_run.rise.CLK OR work_data.input_run.rise_physical.CLK, PT:= , Q=> , ET=> );
IF work_data.input_home.rise.Q AND work_data.can_home THEN
	cut_data.axiss[0].home_done := FALSE;
	cut_data.axiss[1].home_done := FALSE;
	supply_data.axis.home_done := FALSE;
	work_data.state := State.HOME;
END_IF
IF work_data.input_stop.fall_physical.CLK AND NOT work_data.overload.on THEN
	IF work_data.run_auto.timer.Q THEN
		work_data.run_auto.on := TRUE;
	END_IF
	CASE work_data.state OF
		State.RST_DONE:
			IF work_data.input_run.rise.Q OR work_data.input_run.rise_physical.Q THEN
				work_data.state := State.HOME;
			END_IF
		State.READY:
			IF work_data.can_run AND supply_data.state_ready AND cut_data.state = State.READY THEN
				IF (work_data.input_run.timer.Q OR work_data.run_auto.on OR work_data.final_cycle_flag) AND cut_data.state_spindle = State.RUN_ING THEN
					IF work_data.final_cycle_flag THEN
						work_data.final_cycle_flag := FALSE;
						work_data.final_cycle := TRUE;
					END_IF
					work_data.state := State.RUN;
				END_IF
			END_IF
		ELSE
			IF work_data.run_auto.on AND (work_data.input_run.rise.Q OR work_data.input_run.rise_physical.Q) THEN
				work_data.run_auto.on := FALSE;
				work_data.final_cycle_flag := TRUE;
			END_IF
	END_CASE
END_IF
work_data.overload.rise(CLK:= work_data.overload, Q=> );
IF (work_data.input_stop.rise.Q OR work_data.input_stop.fall_physical.Q OR work_data.overload.rise.Q) AND work_data.can_stop THEN
	hmi.jog_micro_per_sec_or_rev := 0;
	work_data.run_auto.on := FALSE;
	work_data.state := State.RST;
END_IF
IF supply_data.input_air AND supply_data.input_hydraulic AND work_data.supply_test_timer.Q THEN
	CASE supply_data.state OF
		State.READY:
			supply_data.state := State.RUN;
		110:
			supply_data.state := 111;
		120:
			supply_data.state := 121;
		130:
			supply_data.state := 131;
		140:
			supply_data.state := State.RUN;
	END_CASE
END_IF
IF supply_data.foil_stuck.on THEN
	IF (supply_data.state = 110 OR supply_data.state = 140) AND supply_data.foil_stuck.fix_rise.Q THEN
		supply_data.state := State.RUN; // run extract foil
	END_IF
	IF supply_data.state = 110 AND supply_data.foil_stuck.fix_timer.Q THEN
		supply_data.state := 111;
	END_IF
END_IF
IF work_data.manual_active THEN
	IF cut_data.state_spindle = State.READY AND work_data.cut_spindle_run_timer.Q THEN
		cut_data.state_spindle := State.RUN;
	END_IF
	IF cut_data.state_spindle >= State.RUN AND work_data.cut_spindle_run_rise.Q THEN
		cut_data.state_spindle := State.RST;
	END_IF
	IF NOT supply_data.hydraulic THEN
		IF work_data.supply_hydraulic_timer.Q THEN
			supply_data.hydraulic := TRUE;
		END_IF
	ELSE
		IF work_data.supply_hydraulic_rise.Q THEN
			supply_data.hydraulic := FALSE;
		END_IF
	END_IF
	IF work_data.input_run.rise.Q OR work_data.input_run.rise_physical.Q THEN
		IF supply_data.state = 110 OR supply_data.state = 120 OR supply_data.state = 130 THEN
			supply_data.state := 141;
		END_IF
		IF supply_data.state = 140 THEN
			supply_data.state := State.READY;
		END_IF
	END_IF
	IF supply_data.state = State.READY THEN
		supply_data.arm_clamp_holder.on := hmi.supply_arm_clamp_holder;
		supply_data.arm_clamp.on := hmi.supply_arm_clamp;
		supply_data.spindle_clamp.on := hmi.supply_spindle_clamp;
		supply_data.spindle_extract.on := hmi.supply_spindle_extract;
	ELSE
		hmi.supply_arm_clamp_holder := supply_data.arm_clamp_holder.on;
		hmi.supply_arm_clamp := supply_data.arm_clamp.on;
		hmi.supply_spindle_clamp := supply_data.spindle_clamp.on;
		hmi.supply_spindle_extract := supply_data.spindle_extract.on;
	END_IF
ELSE
	hmi.supply_arm_clamp_holder := supply_data.arm_clamp_holder.on;
	hmi.supply_arm_clamp := supply_data.arm_clamp.on;
	hmi.supply_spindle_clamp := supply_data.spindle_clamp.on;
	hmi.supply_spindle_extract := supply_data.spindle_extract.on;
END_IF
//
supply_data.arm_clamp_holder.n_timer(IN:= NOT supply_data.arm_clamp_holder.on, PT:= , Q=> , ET=> );
supply_data.arm_clamp_holder.p_timer(IN:= supply_data.arm_clamp_holder.on, PT:= , Q=> , ET=> );
supply_data.arm_clamp.n_timer(IN:= NOT supply_data.arm_clamp.on, PT:= , Q=> , ET=> );
supply_data.arm_clamp.p_timer(IN:= supply_data.arm_clamp.on, PT:= , Q=> , ET=> );
supply_data.spindle_clamp.n_timer(IN:= NOT supply_data.spindle_clamp.on, PT:= , Q=> , ET=> );
supply_data.spindle_clamp.p_timer(IN:= supply_data.spindle_clamp.on, PT:= , Q=> , ET=> );
supply_data.spindle_extract.n_timer(IN:= NOT supply_data.spindle_extract.on, PT:= , Q=> , ET=> );
supply_data.spindle_extract.p_timer(IN:= supply_data.spindle_extract.on, PT:= , Q=> , ET=> );
//////////
//OUTPUT//
//////////
supply_data.spindle_clamp_release := (NOT supply_data.spindle_clamp.on AND NOT supply_data.spindle_clamp.n_timer.Q);
work_data.alarm := work_data.overload.on OR supply_data.foil_stuck.on;
%QX0.0 := supply_data.spindle_clamp.on; // relay 1
%QX0.1 := supply_data.spindle_clamp_release; // relay 2
%QX0.2 := supply_data.hydraulic; // relay 3
%QX0.3 := supply_data.arm_clamp_holder.on; // relay 4
%QX0.4 := cut_data.spindle;
//empty %QX0.5
//empty %QX0.6
//empty %QX0.7
%QX1.0 := supply_data.arm_clamp.on; // relay 5
%QX1.1 := supply_data.spindle_extract.on; // relay 6
%QX1.2 := work_data.alarm; // relay 7
%QX1.3 := FALSE; // relay 8
//empty %QX1.4;
//empty %QX1.5;
//empty %QX1.6;
//empty %QX1.7
//////////
//HMI UP//
//////////
IF hmi.hmi_ready THEN
	hmi.view_input[0] := work_data.input_run.rise_physical.CLK;
	hmi.view_input[1] := work_data.input_stop.fall_physical.CLK;
	hmi.view_input[2] := supply_data.input_air;
	hmi.view_input[3] := supply_data.input_hydraulic;
	hmi.view_input[4] := supply_data.input_arm_clamp_holder_p;
	hmi.view_input[5] := supply_data.input_feeder_small;
	hmi.view_input[6] := supply_data.input_feeder_big;
	hmi.view_input[7] := %IX0.0;
	hmi.view_input[8] := %IX0.1;
	hmi.view_input[9] := %IX1.0;
	hmi.view_input[10] := %IX1.1;
	hmi.view_input[11] := %IX0.4;
	hmi.view_input_jog_index := work_data.input_jog_index;
	hmi.view_input_jog_micro := LREAL_TO_DINT(work_data.jog_encoder^.fActPosition * 1000);
	//
	hmi.view_output[0] := supply_data.arm_clamp_holder.on;
	hmi.view_output[1] := supply_data.arm_clamp.on;
	hmi.view_output[2] := supply_data.spindle_clamp_release;
	hmi.view_output[3] := supply_data.spindle_clamp.on;
	hmi.view_output[4] := supply_data.spindle_extract.on;
	hmi.view_output[5] := supply_data.hydraulic;
	hmi.view_output[6] := work_data.alarm;
	hmi.view_output[7] := cut_data.spindle;
	//
	hmi.view_can_run := work_data.can_run;
	hmi.view_can_stop := work_data.can_stop;
	hmi.view_can_home := work_data.can_home;
	hmi.view_auto := work_data.run_auto.on;
	hmi.view_manual := work_data.manual_active;
	//
	hmi.view_problem[0] := work_data.overload.on;
	hmi.view_problem[1] := supply_data.foil_stuck.on;
	hmi.view_cycle_count := cycle_count;
	hmi.view_cycle_time_msec := work_data.cycle_time_msec;
	//
	hmi.view_axis_micro[0] := LREAL_TO_UDINT(cut_data.axiss[0].ref^.fActPosition);
	hmi.view_axis_micro[1] := LREAL_TO_UDINT(cut_data.axiss[1].ref^.fActPosition);
	hmi.view_axis_micro[2] := LREAL_TO_UDINT(supply_data.axis.ref^.fActPosition);
	hmi.view_axis_mNm[0] := LREAL_TO_UDINT(cut_data.axiss[0].torque_Nm_abs * 1E3);
	hmi.view_axis_mNm[1] := LREAL_TO_UDINT(cut_data.axiss[1].torque_Nm_abs * 1E3);
	hmi.view_axis_mNm[2] := LREAL_TO_UDINT(supply_data.axis.torque_Nm_abs * 1E3);
	//
	hmi.view_cut_spindle_run_ing := cut_data.state_spindle = State.RUN_ING;
	hmi.view_cut_spindle_rpm := LREAL_TO_UDINT(ABS(cut_data.spindle_rps * 60));
	hmi.view_supply_test[0] := (work_data.can_run OR work_data.manual_active) AND supply_data.state_ready;
	hmi.view_supply_test[1] := (work_data.can_run OR work_data.manual_active) AND supply_data.state = 110;
	hmi.view_supply_test[2] := (work_data.can_run OR work_data.manual_active) AND supply_data.state = 120;
	hmi.view_supply_test[3] := (work_data.can_run OR work_data.manual_active) AND supply_data.state = 130;
	//
	hmi.view_state[0] := work_data.state;
	hmi.view_state[1] := supply_data.state;
	hmi.view_state[2] := cut_data.state;
	hmi.view_state[3] := cut_data.state_spindle;
END_IF
END_ACTION

ACTION motion:
FOR i := 0 TO c_axis_i_max BY 1 DO
	axiss_read[i](
		xExecute:= , 
		xAbort:= , 
		uiIndex:= , 
		usiSubIndex:= , 
		Axis:= axiss[i]^, 
		xDone=> , 
		xBusy=> , 
		xError=> , 
		usiDataLength=> , 
		dwValue=> , 
		dwErrorCode=> , 
		eError=> );
	axiss_write[i](
		xExecute:= , 
		xAbort:= , 
		uiIndex:= , 
		usiSubIndex:= , 
		usiDataLength:= , 
		dwValue:= , 
		Axis:= axiss[i]^, 
		xDone=> , 
		xBusy=> , 
		xError=> , 
		dwErrorCode=> , 
		eError=> );
	axiss_read_status[i](
		Axis:= axiss[i]^, 
		Enable:= , 
		Valid=> , 
		Busy=> , 
		Error=> , 
		ErrorID=> , 
		Disabled=> , 
		Errorstop=> , 
		Stopping=> , 
		StandStill=> , 
		DiscreteMotion=> , 
		ContinuousMotion=> , 
		SynchronizedMotion=> , 
		Homing=> , 
		ConstantVelocity=> , 
		Accelerating=> , 
		Decelerating=> , 
		FBErrorOccured=> );
	axiss_set_mode[i](
		Axis:= axiss[i]^, 
		bExecute:= , 
		nControllerMode:= , 
		bDone=> , 
		bBusy=> , 
		bError=> , 
		nErrorID=> );
	axiss_power[i](
		Axis:= axiss[i]^,
		Enable:= , 
		bRegulatorOn:= , 
		bDriveStart:= , 
		Status=> , 
		bRegulatorRealState=> , 
		bDriveStartRealState=> , 
		Busy=> , 
		Error=> , 
		ErrorID=> );
	axiss_reset[i](
		Axis:= axiss[i]^,
		Execute:= ,
		Done=> ,
		Busy=> ,
		Error=> ,
		ErrorID=> );
	axiss_stop[i](
		Axis:= axiss[i]^, 
		Execute:= , 
		Deceleration:= , 
		Jerk:= , 
		Done=> , 
		Busy=> , 
		Error=> , 
		ErrorID=> );
	axiss_inch[i](
		Axis:= axiss[i]^, 
		InchForward:= , 
		InchBackward:= , 
		Distance:= , 
		Velocity:= , 
		Acceleration:= , 
		Deceleration:= , 
		Jerk:= , 
		Busy=> , 
		CommandAborted=> , 
		Error=> , 
		ErrorId=> );
	axiss_fsv[i](
		Axis:= axiss[i]^, 
		bExecute:= , 
		bAbort:= , 
		dwValueMask:= , 
		fSetPosition:= , 
		fSetVelocity:= , 
		fSetAcceleration:= , 
		fSetJerk:= , 
		fSetTorque:= , 
		fSetCurrent:= , 
		bBusy=> , 
		bCommandAborted=> , 
		bError=> , 
		iErrorID=> );
	axiss_sp[i](
		Axis:= axiss[i]^, 
		Execute:= , 
		Position:= , 
		Mode:= , 
		Done=> , 
		Busy=> , 
		Error=> , 
		ErrorID=> );
	axiss_mabs[i](
		Axis:= axiss[i]^, 
		Execute:= , 
		Position:= , 
		Velocity:= , 
		Acceleration:= , 
		Deceleration:= , 
		Jerk:= , 
		Direction:= , 
		BufferMode:= , 
		Done=> , 
		Busy=> , 
		Active=> , 
		CommandAborted=> , 
		Error=> , 
		ErrorID=> );
END_FOR
END_ACTION

ACTION save_check:
hmi.sv_need := (
	save.home_encoder_value_recorded <> hmi.sv.home_encoder_value_recorded OR
	save.max_micro_recorded <> hmi.sv.max_micro_recorded OR
	//
	save.cut_begin_micro[0] <> hmi.sv.cut_begin_micro[0] OR
	save.cut_begin_micro[1] <> hmi.sv.cut_begin_micro[1] OR
	save.cut_rapid_micro[0] <> hmi.sv.cut_rapid_micro[0] OR
	save.cut_rapid_micro[1] <> hmi.sv.cut_rapid_micro[1] OR
	save.cut_end_micro[0] <> hmi.sv.cut_end_micro[0] OR
	save.cut_end_micro[1] <> hmi.sv.cut_end_micro[1] OR
	save.cut_offset_micro[0] <> hmi.sv.cut_offset_micro[0] OR
	save.cut_offset_micro[1] <> hmi.sv.cut_offset_micro[1] OR
	//
	save.cut_lag_micro <> hmi.sv.cut_lag_micro OR
	save.cut_rapid_micro_per_rev <> hmi.sv.cut_rapid_micro_per_rev OR
	save.cut_micro_per_rev <> hmi.sv.cut_micro_per_rev OR
	save.cut_dwell_msec <> hmi.sv.cut_dwell_msec OR
	save.cut_retract_micro <> hmi.sv.cut_retract_micro OR
	save.cut_retract_micro_per_sec <> hmi.sv.cut_retract_micro_per_sec OR
	save.cut_spindle_encoder_resolution <> hmi.sv.cut_spindle_encoder_resolution OR
	//
	save.supply_begin_micro <> hmi.sv.supply_begin_micro OR
	save.supply_mid_micro <> hmi.sv.supply_mid_micro OR
	save.supply_end_micro <> hmi.sv.supply_end_micro OR
	save.supply_micro_per_sec <> hmi.sv.supply_micro_per_sec
);
FOR i := 0 TO c_cylinder_i_max BY 1 DO
	hmi.sv_need := (hmi.sv_need OR
		save.cylinder_n_delay_msec[i] <> hmi.sv.cylinder_n_delay_msec[i] OR
		save.cylinder_p_delay_msec[i] <> hmi.sv.cylinder_p_delay_msec[i]
	);
END_FOR
FOR i := 0 TO c_axis_i_max BY 1 DO
	hmi.sv_need := (hmi.sv_need OR
		save.max_rpm[i] <> hmi.sv.max_rpm[i] OR
		save.gear_dir[i] <> hmi.sv.gear_dir[i] OR
		save.gear_num[i] <> hmi.sv.gear_num[i] OR
		save.gear_den[i] <> hmi.sv.gear_den[i] OR
		save.home_torque_mNm[i] <> hmi.sv.home_torque_mNm[i] OR
		save.home_encoder_value[i] <> hmi.sv.home_encoder_value[i] OR
		save.max_micro[i] <> hmi.sv.max_micro[i] OR
		save.overload_hold_torque_factor[i] <> hmi.sv.overload_hold_torque_factor[i] OR
		save.overload_hold_torque_time_msec[i] <> hmi.sv.overload_hold_torque_time_msec[i] OR
		save.overload_instant_torque_factor[i] <> hmi.sv.overload_instant_torque_factor[i] OR
		save.ramp_time_msec[i] <> hmi.sv.ramp_time_msec[i] OR
		save.jerk_factor[i] <> hmi.sv.jerk_factor[i]
	);
END_FOR
END_ACTION

ACTION save_apply:
///////////
//LIMIT 1//
///////////
FOR i := 0 TO c_cylinder_i_max DO
	save.cylinder_n_delay_msec[i] := MAX(0_100, MIN(5_000, save.cylinder_n_delay_msec[i]));
	save.cylinder_p_delay_msec[i] := MAX(0_100, MIN(5_000, save.cylinder_p_delay_msec[i]));
END_FOR
FOR i := 0 TO c_axis_i_max BY 1 DO
	save.max_rpm[i] := MAX(1000, MIN(axiss_max_rpm[i] - 200, save.max_rpm[i]));
	save.gear_num[i] := MAX(1, save.gear_num[i]);
	save.gear_den[i] := MAX(1, save.gear_den[i]);
	save.home_torque_mNm[i] := MAX(0_100, MIN(LREAL_TO_UINT(axiss_rated_torque_Nm[i] * 1E3), save.home_torque_mNm[i]));
	save.home_encoder_value[i] := MAX(0, MIN(axiss_encoder_resolution[i] - 1, save.home_encoder_value[i]));
	save.max_micro[i] := MAX(10_000, save.max_micro[i]);
	save.overload_hold_torque_factor[i] := MAX(0_010, MIN(3_000, save.overload_hold_torque_factor[i]));
	save.overload_hold_torque_time_msec[i] := MAX(0_010, MIN(2_000, save.overload_hold_torque_time_msec[i]));
	save.overload_instant_torque_factor[i] := MAX(0_010, MIN(3_000, save.overload_instant_torque_factor[i]));
	save.ramp_time_msec[i] := MAX(0_050, MIN(0_800, save.ramp_time_msec[i]));
	save.jerk_factor[i] := MAX(5, MIN(80, save.jerk_factor[i]));
END_FOR
///////////
//APPLY 1//
///////////
FOR i := 0 TO c_axis_i_max BY 1 DO
	CASE i OF
		0: axis_ec_i := ADR(cut_data.axiss[0]);
		1: axis_ec_i := ADR(cut_data.axiss[1]);
		2: axis_ec_i := ADR(supply_data.axis);
	END_CASE
	axis_ec_i^.home_encoder_value_recorded := save.home_encoder_value_recorded;
	axis_ec_i^.home_encoder_value_save := ADR(save.home_encoder_value[i]);
	axis_ec_i^.max_μ_recorded := save.max_micro_recorded;
	axis_ec_i^.max_μ_save := ADR(save.max_micro[i]);
	axis_ec_i^.max_μ := DINT_TO_LREAL(axis_ec_i^.max_μ_save^);
	axis_ec_i^.max_μ_per_sec := axiss_max_μ_per_sec[i];
	axis_ec_i^.home_torque_Nm := UINT_TO_LREAL(save.home_torque_mNm[i]) * 1E-3;
	axis_ec_i^.home_hit_timer.PT := INT_TO_TIME(1_000);
	axis_ec_i^.home_offset_absolute_μ := 5_000;
	axis_ec_i^.home_back_μ_per_sec := MIN(10_000, axis_ec_i^.max_μ_per_sec);
	axis_ec_i^.home_forward_μ_per_sec := MIN(30_000, axis_ec_i^.max_μ_per_sec);
	axis_ec_i^.overload_hold_torque_Nm := axis_ec_i^.torque_rated_Nm * save.overload_hold_torque_factor[i] * 1E-3;
	axis_ec_i^.overload_hold_torque_timer.PT := UINT_TO_TIME(save.overload_hold_torque_time_msec[i]);
	axis_ec_i^.overload_instant_torque_Nm := axis_ec_i^.torque_rated_Nm * save.overload_instant_torque_factor[i] * 1E-3;
	axis_ec_i^.ramp_time_sec := UINT_TO_LREAL(save.ramp_time_msec[i]) * 1E-3;
	axis_ec_i^.jerk_factor := save.jerk_factor[i];
END_FOR
///////////
//LIMIT 2//
///////////
FOR i := 0 TO 1 DO
	save.cut_end_micro[i] := MAX(10_000, MIN(save.max_micro[i], save.cut_end_micro[i]));
	save.cut_rapid_micro[i] := MIN(save.cut_end_micro[i] - 0_500, save.cut_rapid_micro[i]);
	save.cut_begin_micro[i] := MIN(save.cut_rapid_micro[i] - 0_500, save.cut_begin_micro[i]);
	save.cut_offset_micro[i] := MAX(-9_000, MIN(9_000, save.cut_offset_micro[0]));
END_FOR
//
save.cut_lag_micro := MAX(0_100, MIN(3_000, save.cut_lag_micro));
save.cut_rapid_micro_per_rev := MAX(0_001, MIN(1_000, save.cut_rapid_micro_per_rev));
save.cut_micro_per_rev := MAX(0_001, MIN(0_500, save.cut_micro_per_rev));
save.cut_dwell_msec := MAX(0_001, MIN(1_000, save.cut_dwell_msec));
save.cut_retract_micro_per_sec := MAX(5_000, MIN(LREAL_TO_UDINT(cut_data.axiss[0].max_μ_per_sec), save.cut_retract_micro_per_sec));
//
save.home_encoder_value[0] := MAX(0, MIN(cut_data.axiss[0].encoder_resolution - 1, save.home_encoder_value[0]));
save.home_encoder_value[1] := MAX(0, MIN(cut_data.axiss[1].encoder_resolution - 1, save.home_encoder_value[1]));
save.home_encoder_value[2] := MAX(0, MIN(supply_data.axis.encoder_resolution - 1, save.home_encoder_value[2]));
///////////
//APPLY 2//
///////////
cut_data.lag_μm := UDINT_TO_LREAL(save.cut_lag_micro);
cut_data.rapid_μm_per_rev := UDINT_TO_LREAL(save.cut_rapid_micro_per_rev);
cut_data.μm_per_rev := UDINT_TO_LREAL(save.cut_micro_per_rev);
cut_data.dwell_timer.PT := UINT_TO_TIME(save.cut_dwell_msec);
cut_data.retract_μm := UDINT_TO_LREAL(save.cut_retract_micro);
cut_data.retract_μm_per_sec := UDINT_TO_LREAL(save.cut_retract_micro_per_sec);
cut_data.spindle_encoder_resolution := MAX(1, save.cut_spindle_encoder_resolution);
//
FOR i := 0 TO c_cylinder_i_max DO
	CASE i OF
		0: cylinder_i := ADR(supply_data.arm_clamp_holder);
		1: cylinder_i := ADR(supply_data.arm_clamp);
		2: cylinder_i := ADR(supply_data.spindle_clamp);
		3: cylinder_i := ADR(supply_data.spindle_extract);
	END_CASE
	cylinder_i^.n_timer.PT := UINT_TO_TIME(save.cylinder_n_delay_msec[i]);
	cylinder_i^.p_timer.PT := UINT_TO_TIME(save.cylinder_p_delay_msec[i]);
END_FOR
//
supply_data.foil_stuck.timer.PT := INT_TO_TIME(1_000);
supply_data.foil_stuck.fix_timer.PT := INT_TO_TIME(1_000);
//
work_data.input_run.timer.PT := INT_TO_TIME(0_300);
work_data.run_auto.timer.PT := INT_TO_TIME(3_000);
work_data.cut_spindle_run_timer.PT := INT_TO_TIME(1_000);
work_data.supply_test_timer.PT := INT_TO_TIME(0_300);
work_data.supply_hydraulic_timer.PT := INT_TO_TIME(0_300);
/////////
//FINAL//
/////////
hmi.sv := save;
END_ACTION

ACTION work:
CASE work_data.state OF
	State.RST:
		supply_data.axis.overload_check := FALSE;
		cut_data.axiss[0].overload_check := FALSE;
		cut_data.axiss[1].overload_check := FALSE;
		supply_data.state := State.RST;
		cut_data.state := State.RST;
		cut_data.state_spindle := State.RST;
		work_data.jog_encoder_counter_set.xExecute := TRUE;
		work_data.manual_active := FALSE;
		work_data.alarm := FALSE;
		work_data.final_cycle_flag := FALSE;
		work_data.final_cycle := FALSE;
		StateNext(work_data.state);
	2:
		IF (
			supply_data.state = State.RST_DONE AND
			cut_data.state = State.RST_DONE AND
			cut_data.state_spindle = State.READY AND
			work_data.jog_encoder_counter_set.xDone
		) THEN
			work_data.state := State.RST_DONE;
		END_IF
	State.RST_DONE:
		//do nothing
	//////\\
	////\\\\
	//\\\\\\
	State.HOME:
		cut_data.state := State.HOME;
		StateNext(work_data.state);
	52:
		IF cut_data.state = State.HOME_DONE THEN
			supply_data.state := State.HOME;
			StateNext(work_data.state);
		END_IF
	53:
		IF supply_data.state = State.HOME_DONE THEN
			supply_data.axis.overload_check := TRUE;
			cut_data.axiss[0].overload_check := TRUE;
			cut_data.axiss[1].overload_check := TRUE;
			work_data.state := State.HOME_DONE;
		END_IF
	//
	State.HOME_DONE:
		supply_data.state := State.HOME_OFFSET;
		cut_data.state := State.HOME_OFFSET;
		StateNext(work_data.state);
	91:
		IF (
			supply_data.state = State.HOME_OFFSET_DONE AND
			cut_data.state = State.HOME_OFFSET_DONE
		) THEN
			work_data.state := State.HOME_OFFSET_DONE;
		END_IF
	State.HOME_OFFSET_DONE:
		supply_data.state := State.READY;
		cut_data.state := State.READY;
		work_data.state := State.READY;
		work_data.manual_active := TRUE;
		IF NOT save.home_encoder_value_recorded THEN
			save.home_encoder_value_recorded := TRUE;
			save_apply();
		END_IF
	//////\\
	////\\\\
	//\\\\\\
	State.READY:
		IF work_data.manual_active THEN
			CASE work_data.input_jog_index OF
				0: work_data.jog_i := ADR(cut_data.axiss[0]);
				1: work_data.jog_i := ADR(cut_data.axiss[1]);
				2: work_data.jog_i := ADR(supply_data.axis);
			END_CASE
			work_data.jog_i^.jog_delta := hmi.jog_micro_per_sec_or_rev * (work_data.jog_encoder^.fActPosition - work_data.jog_encoder_last);
			work_data.jog_i^.jog_velocity := hmi.jog_micro_per_sec_or_rev * work_data.jog_encoder^.fActVelocity;
			work_data.jog_i^.jog_acceleration := hmi.jog_micro_per_sec_or_rev * work_data.jog_encoder^.fActAcceleration;
			work_data.jog_encoder_last := work_data.jog_encoder^.fActPosition;
		END_IF
	//////\\
	////\\\\
	//\\\\\\
	State.RUN:
		IF supply_data.state_ready AND cut_data.state_spindle = State.RUN_ING THEN
			work_data.manual_active := FALSE;
			supply_data.state := State.RUN;
			work_data.cycle_start_msec := time_msec;
			StateNext(work_data.state);
		END_IF
	102:
		IF supply_data.state = 110 THEN
			supply_data.state := 111;
			StateNext(work_data.state);
		END_IF
	103:
		IF supply_data.foil_stuck.on THEN
			work_data.alarm := TRUE;
		END_IF
		IF supply_data.state = 120 THEN
			cut_data.state := State.RUN;
			IF work_data.final_cycle THEN
				work_data.final_cycle := FALSE;
				supply_data.state := 141;
				work_data.state := 121;
			ELSE
				supply_data.state := 121;
				work_data.state := 111;
			END_IF
		END_IF
	//normal cycle
	111:
		IF supply_data.state = 130 THEN
			supply_data.state := 131;
			StateNext(work_data.state);
		END_IF
	112:
		IF cut_data.state = State.READY AND supply_data.state = 140 THEN
			work_data.state := 131;
		END_IF
	//final cycle
	121:
		IF cut_data.state = State.READY AND supply_data.state = 140 THEN
			supply_data.state := State.RUN; // extract foil
			StateNext(work_data.state);
		END_IF
	122:
		IF supply_data.state = 110 THEN
			supply_data.state := State.READY; // ready for rerun
			work_data.state := 131;
		END_IF
	//end
	131:
		work_data.state := State.READY;
		work_data.cycle_time_msec := ULINT_TO_UDINT(time_msec - work_data.cycle_start_msec);
		work_data.alarm := FALSE;
		IF (time_msec - cycle_count_reset_time_msec) > 86400_000 THEN
			cycle_count := 0;
			cycle_count_reset_time_msec := (time_msec / 86400_000) * 86400_000;
		END_IF
		cycle_count := cycle_count + 1;
END_CASE
END_ACTION

END_PROGRAM

// Device/Application/StateNext
FUNCTION StateNext
VAR_INPUT
	state: REFERENCE TO INT;
END_VAR
VAR
END_VAR

state := state + 1;

END_FUNCTION

// Device/Application/SupplyFB
FUNCTION_BLOCK SupplyFB
VAR_INPUT
	d: POINTER TO SupplyData;
END_VAR

////////
//MAIN//
////////
d^.state_ready := d^.state = State.READY OR d^.state = 140;
d^.axis_fb(d:= ); // data của hàm này đã được set ở hàm MAIN
d^.foil_stuck.timer(IN:= , PT:= , Q=> , ET=> );
d^.arm_clamp_holder_p_rise(CLK:= d^.input_arm_clamp_holder_p, Q=> );
CASE d^.state OF
	//////\\
	////\\\\
	//\\\\\\
	State.RST:
		d^.arm_clamp_holder.on := FALSE;
		d^.spindle_extract.on := FALSE;
		d^.foil_stuck.on := FALSE;
		StateNext(d^.state);
	2:
		IF (
			d^.arm_clamp_holder.n_timer.Q AND
			d^.spindle_extract.n_timer.Q
		) THEN
			d^.axis.state := State.RST;
			StateNext(d^.state);
		END_IF
	3:
		IF d^.axis.state = State.RST_DONE THEN
			d^.state := State.RST_DONE;
		END_IF
	//////\\
	////\\\\
	//\\\\\\
	State.HOME:
		d^.arm_clamp.on := FALSE;
		d^.spindle_clamp.on := FALSE;
		StateNext(d^.state);
	52:
		IF (
			d^.arm_clamp.n_timer.Q AND
			d^.spindle_clamp.n_timer.Q
		) THEN
			d^.axis.state := State.HOME;
			StateNext(d^.state);
		END_IF
	53:
		IF d^.axis.state = State.HOME_DONE THEN
			d^.state := State.HOME_DONE;
		END_IF
	//////\\
	////\\\\
	//\\\\\\
	State.HOME_OFFSET:
		d^.axis.home_offset_μ := d^.begin_μdeg;
		d^.axis.state := State.HOME_OFFSET;
		StateNext(d^.state);
	92:
		IF d^.axis.state = State.HOME_OFFSET_DONE THEN
			d^.axis.state := State.READY;
			d^.state := State.HOME_OFFSET_DONE;
		END_IF
	State.READY:
		//do nothing
	//////\\
	////\\\\
	//\\\\\\
	// thoát phôi
	State.RUN:
		d^.arm_clamp_holder.on := FALSE; // make sure collision free move
		StateNext(d^.state);
	102:
		IF d^.arm_clamp_holder.n_timer.Q THEN
			d^.spindle_clamp.on := FALSE;
			StateNext(d^.state);
		END_IF
	103:
		IF d^.spindle_clamp.n_timer.Q THEN
			d^.spindle_extract.on := TRUE;
			StateNext(d^.state);
		END_IF
	104:
		IF d^.spindle_extract.p_timer.Q THEN
			d^.spindle_extract.on := FALSE;
			StateNext(d^.state);
		END_IF
	105:
		IF d^.spindle_extract.n_timer.Q THEN
			d^.state := 110;
		END_IF
	// cấp phôi
	111:
		d^.arm_clamp_holder.on := FALSE; // make sure collision free move
		d^.foil_stuck.timer.IN := FALSE;
		StateNext(d^.state);
	112:
		IF d^.arm_clamp_holder.n_timer.Q AND d^.axis.state = State.READY THEN
			d^.axis.target_position_μ := d^.end_μdeg;
			d^.axis.target_velocity_μ_per_sec := d^.μdeg_per_sec;
			d^.axis.state := State.RUN;
			StateNext(d^.state);
		END_IF
	113:
		IF d^.axis.state = State.READY THEN
			d^.arm_clamp_holder.on := TRUE;
			d^.foil_stuck.timer.IN := TRUE;
			StateNext(d^.state);
		END_IF
	114:
		IF d^.foil_stuck.timer.Q THEN
			d^.foil_stuck.on := TRUE;
			d^.foil_stuck.timer.IN := FALSE;
			d^.state := 141;
		END_IF
		IF d^.arm_clamp_holder_p_rise.Q THEN
			d^.spindle_clamp.on := TRUE;
			StateNext(d^.state);
		END_IF
	115:
		IF d^.spindle_clamp.p_timer.Q THEN
			d^.arm_clamp.on := FALSE;
			StateNext(d^.state);
		END_IF
	116:
		IF d^.arm_clamp.n_timer.Q THEN
			d^.arm_clamp_holder.on := FALSE;
			StateNext(d^.state);
		END_IF
	117:
		IF d^.arm_clamp_holder.n_timer.Q THEN
			d^.foil_stuck.on := FALSE;
			d^.state := 120;
		END_IF
	// lấy phôi mới
	121:
		d^.arm_clamp_holder.on := FALSE; // make sure collision free move
		StateNext(d^.state);
	122:
		IF d^.arm_clamp_holder.n_timer.Q AND d^.axis.state = State.READY THEN
			d^.axis.target_position_μ := d^.begin_μdeg;
			d^.axis.target_velocity_μ_per_sec := d^.μdeg_per_sec;
			d^.axis.state := State.RUN;
			StateNext(d^.state);
		END_IF
	123:
		IF d^.axis.state = State.READY THEN
			d^.arm_clamp_holder.on := TRUE;
			StateNext(d^.state);
		END_IF
	124:
		IF d^.arm_clamp_holder.p_timer.Q THEN
			d^.arm_clamp.on := TRUE;
			StateNext(d^.state);
		END_IF
	125:
		IF d^.arm_clamp.p_timer.Q THEN
			d^.arm_clamp_holder.on := FALSE;
			StateNext(d^.state);
		END_IF
	126:
		IF d^.arm_clamp_holder.n_timer.Q THEN
			d^.state := 130;
		END_IF
	// di chuyển đến vị trí chờ
	131:
		d^.arm_clamp_holder.on := FALSE; // make sure collision free move
		StateNext(d^.state);
	132:
		IF d^.arm_clamp_holder.n_timer.Q AND d^.axis.state = State.READY THEN
			d^.axis.target_position_μ := d^.mid_μdeg;
			d^.axis.target_velocity_μ_per_sec := d^.μdeg_per_sec;
			d^.axis.state := State.RUN;
			StateNext(d^.state);
		END_IF
	133:
		IF d^.axis.state = State.READY THEN
			d^.state := 140;
		END_IF
	// di chuyển đến vị trí nghỉ
	141:
		d^.arm_clamp_holder.on := FALSE; // make sure collision free move
		StateNext(d^.state);
	142:
		IF d^.arm_clamp_holder.n_timer.Q AND d^.axis.state = State.READY THEN
			d^.axis.target_position_μ := d^.begin_μdeg;
			d^.axis.target_velocity_μ_per_sec := d^.μdeg_per_sec;
			d^.axis.state := State.RUN;
			StateNext(d^.state);
		END_IF
	143:
		IF d^.axis.state = State.READY THEN
			d^.state := 140;
		END_IF
END_CASE

END_FUNCTION_BLOCK

// Device/Application/CutFB
FUNCTION_BLOCK CutFB
VAR_INPUT
	d: POINTER TO CutData;
END_VAR

VAR CONSTANT
	c_stable_cycle_valid: INT := 2;
END_VAR

////////
//MAIN//
////////
d^.axiss_fb[0](d:= ); // data của hàm này đã được set ở hàm MAIN
d^.axiss_fb[1](d:= );
d^.dwell_timer(IN:= , PT:= , Q=> , ET=> );
IF d^.time_msec - d^.spindle_encoder_time_msec_last >= 2_000 THEN
	d^.time_delta_sec := ULINT_TO_LREAL(d^.time_msec - d^.spindle_encoder_time_msec_last) * 1E-3;
	d^.spindle_rps := (
			DINT_TO_LREAL(d^.spindle_encoder_counter.diValue - d^.spindle_encoder_counter_last) / d^.spindle_encoder_resolution
		) / d^.time_delta_sec;
	d^.spindle_rps := MIN(3000 / 60, d^.spindle_rps);
	d^.spindle_encoder_counter_last := d^.spindle_encoder_counter.diValue;
	d^.spindle_encoder_time_msec_last := d^.time_msec;
	IF d^.spindle_rps - d^.spindle_rps_last < 0.5 THEN
		d^.spindle_rps_stable_cycle := MIN(d^.spindle_rps_stable_cycle + 1, c_stable_cycle_valid);
	ELSE
		d^.spindle_rps_stable_cycle := MAX(0, d^.spindle_rps_stable_cycle - 1);
	END_IF
	d^.spindle_rps_last := d^.spindle_rps;
END_IF
CASE d^.state OF
	//////\\
	////\\\\
	//\\\\\\
	State.RST:
		d^.axiss[0].state := State.RST;
		d^.axiss[1].state := State.RST;
		StateNext(d^.state);
	2:
		IF (
			d^.axiss[0].state = State.RST_DONE AND
			d^.axiss[1].state = State.RST_DONE
		)
		THEN
			d^.state := State.RST_DONE;
		END_IF
	//////\\
	////\\\\
	//\\\\\\
	State.HOME:
		d^.axiss[0].state := State.HOME;
		d^.axiss[1].state := State.HOME;
		StateNext(d^.state);
	52:
		IF (
			d^.axiss[0].state = State.HOME_DONE AND
			d^.axiss[1].state = State.HOME_DONE
		) THEN
			d^.state := State.HOME_DONE;
		END_IF
	//////\\
	////\\\\
	//\\\\\\
	State.HOME_OFFSET:
		d^.axiss[0].home_offset_μ := d^.retract_μm;
		d^.axiss[1].home_offset_μ := d^.retract_μm;
		d^.axiss[0].state := State.HOME_OFFSET;
		d^.axiss[1].state := State.HOME_OFFSET;
		StateNext(d^.state);
	92:
		IF (
			d^.axiss[0].state = State.HOME_OFFSET_DONE AND
			d^.axiss[1].state = State.HOME_OFFSET_DONE
		) THEN
			d^.axiss[0].state := State.READY;
			d^.axiss[1].state := State.READY;
			d^.state := State.HOME_OFFSET_DONE;
		END_IF
	//////\\
	////\\\\
	//\\\\\\
	State.READY:
		//do nothing
	//////\\
	////\\\\
	//\\\\\\
	State.RUN:
		IF (
			d^.axiss[0].state = State.READY AND
			d^.axiss[1].state = State.READY
		) THEN
			d^.axiss[0].target_position_μ := d^.retract_μm;
			d^.axiss[0].target_velocity_μ_per_sec := d^.retract_μm_per_sec;
			d^.axiss[0].state := State.RUN;
			d^.axiss[1].target_position_μ := d^.retract_μm;
			d^.axiss[1].target_velocity_μ_per_sec := d^.retract_μm_per_sec;
			d^.axiss[1].state := State.RUN;
			d^.dwell_timer.IN := FALSE;
			StateNext(d^.state);
		END_IF
	102:
		IF (
			d^.axiss[0].state = State.READY AND
			d^.axiss[1].state = State.READY
		) THEN
			d^.axiss[0].target_position_μ := d^.begin_μm[0];
			d^.axiss[0].target_velocity_μ_per_sec := d^.retract_μm_per_sec;
			d^.axiss[0].state := State.RUN;
			d^.axiss[1].target_position_μ := d^.begin_μm[1];
			d^.axiss[1].target_velocity_μ_per_sec := d^.retract_μm_per_sec;
			d^.axiss[1].state := State.RUN;
			StateNext(d^.state);
		END_IF
	103:
		IF (
			d^.axiss[0].state = State.READY AND
			d^.axiss[1].state = State.READY
		) THEN
			d^.axiss[0].target_position_μ := d^.rapid_μm[0]; // đã có giới hạn trong AxisLinearFB nên không cần giới hạn ở đây
			d^.axiss[0].target_velocity_μ_per_sec := d^.rapid_μm_per_rev * d^.spindle_rps;
			d^.axiss[0].state := State.RUN;
			StateNext(d^.state);
		END_IF
	104:
		IF (d^.axiss[0].ref^.fActPosition - d^.begin_μm[0]) >= d^.lag_μm OR d^.axiss[0].state = State.READY THEN
			d^.axiss[1].target_position_μ := d^.rapid_μm[1];
			d^.axiss[1].target_velocity_μ_per_sec := d^.rapid_μm_per_rev * d^.spindle_rps;
			d^.axiss[1].state := State.RUN;
			StateNext(d^.state);
		END_IF
	105:
		IF (
			d^.axiss[0].state = State.READY AND
			d^.axiss[1].state = State.READY
		) THEN
			d^.axiss[0].target_position_μ := d^.end_μm[0];
			d^.axiss[0].target_velocity_μ_per_sec := d^.μm_per_rev * d^.spindle_rps;
			d^.axiss[0].state := State.RUN;
			StateNext(d^.state);
		END_IF
	106:
		IF (d^.axiss[0].ref^.fActPosition - d^.rapid_μm[0]) >= d^.lag_μm OR d^.axiss[0].state = State.READY THEN
			d^.axiss[1].target_position_μ := d^.end_μm[1];
			d^.axiss[1].target_velocity_μ_per_sec := d^.μm_per_rev * d^.spindle_rps;
			d^.axiss[1].state := State.RUN;
			StateNext(d^.state);
		END_IF
	107:
		IF (
			d^.axiss[0].state = State.READY AND
			d^.axiss[1].state = State.READY
		) THEN
			d^.dwell_timer.IN := TRUE;
			StateNext(d^.state);
		END_IF
	108:
		IF d^.dwell_timer.Q THEN
			d^.axiss[0].target_position_μ := d^.retract_μm;
			d^.axiss[0].target_velocity_μ_per_sec := d^.retract_μm_per_sec;
			d^.axiss[0].state := State.RUN;
			d^.axiss[1].target_position_μ := d^.retract_μm;
			d^.axiss[1].target_velocity_μ_per_sec := d^.retract_μm_per_sec;
			d^.axiss[1].state := State.RUN;
			StateNext(d^.state);
		END_IF
	109:
		IF (
			d^.axiss[0].state = State.READY AND
			d^.axiss[1].state = State.READY
		) THEN
			d^.state := State.READY;
		END_IF
END_CASE
///////////
//SPINDLE//
///////////
CASE d^.state_spindle OF
	State.RST:
		d^.spindle := FALSE;
		d^.spindle_rps_stable_cycle := 0;
	 	StateNext(d^.state_spindle);
	2:
		d^.state_spindle := State.READY;
	//////\\
	////\\\\
	//\\\\\\
	State.READY:
		//do nothing
	//////\\
	////\\\\
	//\\\\\\
	State.RUN:
		d^.spindle := TRUE;
		d^.spindle_rps_stable_cycle := 0;
		StateNext(d^.state_spindle);
	102:
		IF d^.spindle_rps > 10 AND d^.spindle_rps_stable_cycle = c_stable_cycle_valid THEN
			d^.state_spindle := State.RUN_ING;
		END_IF
	//////\\
	////\\\\
	//\\\\\\
	State.RUN_ING:
		//check
END_CASE

END_FUNCTION_BLOCK

// Device/Application/AxisFB
FUNCTION_BLOCK PUBLIC AxisFB
VAR_INPUT
	d: POINTER TO AxisEC;
END_VAR

d^.torque_Nm := d^.ref^.fActTorque;
d^.torque_Nm_abs := ABS(d^.torque_Nm);
// giá trị .fActTorque có thể khác nhau tuỳ PLC, trong trường hợp PLC Inovance này fActTorque là giá trị từ phần trăm moment
// 0.0% đến hơn 100.0%, nên phải nhân với .torque_rated_Nm đọc được ở hàm MAIN
d^.home_hit_timer(IN:= , PT:= , Q=> , ET=> );
// timer để lấy gốc, khi lùi về chạm gốc, giá trị moment sẽ tăng lên đến giá trị quy định (trong chương trình này là 1.27Nm)
// để tránh bị nhiễu thì moment quy định cần phải duy trì trong một thời gian mới có thể xác định gốc
d^.overload_hold_torque_timer(IN:= , PT:= , Q=> , ET=> );
// timer quá tải
IF d^.overload_check THEN
	d^.overload_hold_torque_timer.IN := d^.torque_Nm_abs > d^.overload_hold_torque_Nm;
	d^.overload := d^.overload_hold_torque_timer.Q OR d^.torque_Nm_abs > d^.overload_instant_torque_Nm;
END_IF
//////\\
////\\\\
//\\\\\\
d^.set_torque_limit(
	scale_factor:= d^.ref^.fScalefactor, 
	write:= d^.write, 
	torque_rated_Nm:= d^.torque_rated_Nm, 
	negative_Nm:= , 
	positive_Nm:= , 
	execute:= , 
	done=> );
CASE d^.state OF
	State.RST: // reset trục
		d^.read_status^.Enable := TRUE; // bật đọc trạng thái servo
		StateNext(d^.state);
	2:
		IF d^.read_status^.Valid THEN
			StateNext(d^.state);
		END_IF
	3:
		d^.inch^.InchBackward := FALSE;
		d^.inch^.InchForward := FALSE;
		d^.fsv^.bExecute := FALSE;
		d^.fsv^.fSetPosition := d^.ref^.fActPosition;
		d^.set_torque_limit.execute := FALSE;
		StateNext(d^.state);
	4:
		IF NOT d^.inch^.Busy AND NOT d^.fsv^.bError THEN
			StateNext(d^.state);
		END_IF
	5:
		IF d^.mabs^.Busy THEN // nếu hàm dịch chuyển MC_MoveAbsolute đang hoạt dộng thì kích hoạt hàm MC_Stop
			d^.stop^.Deceleration := d^.mabs^.Velocity / 0.01;
			d^.stop^.Jerk := d^.stop^.Deceleration * d^.jerk_factor;
			d^.stop^.Execute := TRUE;
			StateNext(d^.state);
		ELSE // nếu không thì nhảy đến bước tiếp theo
			d^.state := 21;
		END_IF
	6: // hàm SMC_Inch đang không hoạt động và hàm MC_Stop hoàn thành
		IF d^.stop^.Done THEN
			d^.state := 21;
		END_IF
	//
	21:
		d^.mabs^.Execute := FALSE; // sau khi các hàm hoàn thành, phải đặt biến Execute về FALSE
		d^.stop^.Execute := FALSE; // vì muốn chạy hàm cần có tín hiệu rising edge
		d^.power^.bDriveStart := FALSE; // tắt servo
		StateNext(d^.state);
	22:
		IF NOT d^.power^.Status THEN // đã tắt xong servo
			StateNext(d^.state);
		END_IF
	23:
		IF d^.read_status^.FBErrorOccured THEN // nếu có lỗi xảy ra thì xoá lỗi cũ
			SMC_ClearFBError(pDrive:= d^.ref); // xoá lỗi
			StateNext(d^.state);
		ELSE // nếu không có thì nhảy đến bước cuối
			d^.state := 31;
		END_IF
	24:
		IF d^.read_status^.FBErrorOccured THEN
			d^.reset^.Execute := TRUE; // reset lỗi
			StateNext(d^.state);
		END_IF
	25:
		IF d^.reset^.Done THEN
			d^.reset^.Execute := FALSE;
			SMC_ClearFBError(pDrive:= d^.ref); // xoá lỗi
			d^.state := 31;
		END_IF
	//
	31:
		d^.read_status^.Enable := FALSE;
		d^.state := State.RST_DONE;
	//////\\
	////\\\\
	//\\\\\\
	State.HOME:
		d^.power^.bDriveStart := TRUE; // bật servo để bắt đầu lấy gốc
		StateNext(d^.state);
	52:
		IF d^.power^.Status THEN // servo đã sẵn sàng
			StateNext(d^.state);
		END_IF
	53:
		IF d^.home_done THEN // đã lấy gốc trước đó thì nhảy đến bước HOME_FORWARD
			d^.state := State.HOME_FORWARD;
		ELSE // chưa lấy gốc thì qua bước tiếp theo
			IF d^.home_to_encoder THEN
				d^.state := 59;
			ELSE
				StateNext(d^.state);
			END_IF
		END_IF
	54:
		d^.set_mode^.nControllerMode := SMC_CONTROLLER_MODE.SMC_velocity;// chuyển chế độ servo sang tốc độ
		// ở chế độ .SMC_torque hoặc .SMC_velocity, khi servo vị chặn nó sẽ không vọt sau khi được nhả ra
		d^.set_mode^.bExecute := TRUE;
		StateNext(d^.state);
	55:
		IF d^.set_mode^.bDone THEN // chuyển chế độ xong
			d^.set_mode^.bExecute := FALSE;
			StateNext(d^.state);
		END_IF
	56:
		d^.set_torque_limit.negative_Nm := d^.home_torque_Nm;
		d^.set_torque_limit.positive_Nm := d^.home_torque_Nm;
		d^.set_torque_limit.execute := TRUE;
		StateNext(d^.state);
	57:
		IF d^.set_torque_limit.done THEN
			d^.set_torque_limit.execute := FALSE;
			StateNext(d^.state);
		END_IF
	58:
		d^.inch^.Velocity := d^.home_back_μ_per_sec; // lùi về
		d^.inch^.Distance := 1E16;
		d^.inch^.Acceleration := d^.inch^.Velocity / 0.1;
		d^.inch^.Deceleration := d^.inch^.Acceleration;
		d^.inch^.Jerk := d^.inch^.Acceleration * d^.jerk_factor;
		d^.inch^.InchBackward := TRUE; // .InchBackward là lùi
		d^.inch^.InchForward := FALSE; // .InchForward là tiến
		// nếu .InchBackward và .InchForward cùng bằng TRUE hoặc FALSE thì servo không chạy
		d^.home_hit_timer.IN := FALSE; // reset timer
		d^.home_hit_test := FALSE; // reset test
		StateNext(d^.state);
	59:
		d^.home_hit_timer.IN := d^.torque_Nm_abs >= d^.home_torque_Nm * 0.95 OR d^.home_hit_test; // set timer, * 0.95 để chắc ăn, tránh bị nhiễu
		IF d^.home_hit_timer.Q OR d^.home_to_encoder THEN // khi timer kích hoạt, dừng hàm SMC_Inch
			d^.inch^.InchBackward := FALSE;
			d^.inch^.InchForward := FALSE;
			d^.mabs^.Position := d^.ref^.fActPosition + d^.home_offset_absolute_μ;
			IF d^.home_encoder_value_recorded THEN
				calculate_home_delta_μ();
				d^.mabs^.Position := d^.mabs^.Position + d^.home_delta_μ;
			ELSE
				d^.home_encoder_value_save^ := d^.encoder_single_position;
				d^.home_encoder_value_recorded := TRUE;
			END_IF
			// gán tạm giá trị vào hàm MC_MoveAbsolute để đến bước tiếp theo
			// .fActPosition là vị trí thực tế của servo
			// ví dụ .fActPosition khi chạm là -123_000, có thể dùng "_" để phân cách các con số cho dễ đọc
			// .home_offset_absolute_micron = 1_000
			// d^.mabs^.Position sẽ bằng -123_000 + 1_000 = -122_000
			StateNext(d^.state);
		END_IF
	60:
		d^.sp^.Position := d^.ref^.fActPosition - d^.mabs^.Position;
		// thực hiện hàm MC_SetPosition để đưa giá trị .fActPosition về 0
		// bây giờ giá trị d^.sp^.Position = -123_000 - (-122_000) = -1_000
		// bây giờ servo đang ở vị trí va chạm, để về gốc thì nó phải dịch chuyển 1_000 micron
		// vậy vị trí gốc cách vị trí va chạm đúng bằng .home_offset_absolute_micron
		d^.sp^.Execute := TRUE;
		StateNext(d^.state);
	61:
		IF d^.sp^.Done THEN
			d^.sp^.Execute := FALSE;
			IF d^.max_μ_recorded THEN // đã có chiều dài trục -> tiến tới HOME_FORWARD
				d^.state := State.HOME_FORWARD;
			ELSE
				StateNext(d^.state); // tìm chiều dài trục
			END_IF
		END_IF
	62:
		d^.inch^.Velocity := d^.home_back_μ_per_sec; // tiến tới
		d^.inch^.Distance := 1E16;
		d^.inch^.Acceleration := d^.inch^.Velocity / 0.1;
		d^.inch^.Deceleration := d^.inch^.Acceleration;
		d^.inch^.Jerk := d^.inch^.Acceleration * d^.jerk_factor;
		d^.inch^.InchBackward := FALSE; // .InchBackward là lùi
		d^.inch^.InchForward := TRUE; // .InchForward là tiến
		// nếu .InchBackward và .InchForward cùng bằng TRUE hoặc FALSE thì servo không chạy
		d^.home_hit_timer.IN := FALSE; // reset timer
		d^.home_hit_test := FALSE; // reset test
		StateNext(d^.state);
	63:
		d^.home_hit_timer.IN := d^.torque_Nm_abs >= d^.home_torque_Nm * 0.95 OR d^.home_hit_test; // set timer, * 0.95 để chắc ăn, tránh bị nhiễu
		IF d^.home_hit_timer.Q THEN // khi timer kích hoạt, dừng hàm SMC_Inch
			d^.inch^.InchBackward := FALSE;
			d^.inch^.InchForward := FALSE;
			d^.max_μ := d^.ref^.fActPosition - d^.home_offset_absolute_μ;
			d^.max_μ_save^ := LREAL_TO_DINT(d^.max_μ);
			d^.max_μ_recorded := TRUE;
			d^.state := State.HOME_FORWARD;
		END_IF
	//////\\
	////\\\\
	//\\\\\\
	State.HOME_FORWARD:
		IF NOT d^.inch^.Busy THEN
			d^.set_mode^.nControllerMode := SMC_CONTROLLER_MODE.SMC_position; // set mode về điều khiển vị trí
			d^.set_mode^.bExecute := TRUE;
			StateNext(d^.state);
		END_IF
	72:
		IF d^.set_mode^.bDone THEN
			d^.set_mode^.bExecute := FALSE;
			StateNext(d^.state);
		END_IF
	73:
		// đưa giới hạn moment về 300%
		d^.set_torque_limit.negative_Nm := d^.torque_rated_Nm * 3.0;
		d^.set_torque_limit.positive_Nm := d^.torque_rated_Nm * 3.0;
		d^.set_torque_limit.execute := TRUE;
		StateNext(d^.state);
	74:
		IF d^.set_torque_limit.done THEN
			d^.set_torque_limit.execute := FALSE;
			StateNext(d^.state);
		END_IF
	75:
		// dịch chuyển tới vị trí gốc
		IF d^.home_done AND d^.home_done_forward_ignore THEN
			d^.mabs^.Position := d^.ref^.fActPosition;
		ELSE
			d^.mabs^.Position := 0;
		END_IF
		d^.mabs^.Velocity := d^.home_forward_μ_per_sec;
		d^.mabs^.Acceleration := d^.mabs^.Velocity / d^.ramp_time_sec;
		d^.mabs^.Deceleration := d^.mabs^.Acceleration;
		d^.mabs^.Jerk := d^.mabs^.Acceleration * d^.jerk_factor;
		d^.mabs^.Direction := MC_DIRECTION.shortest; // nếu là trục module, di chuyển đến vị trí gần nhất
		d^.mabs^.Execute := TRUE;
		StateNext(d^.state);
	76:
		IF d^.mabs^.Done THEN
			d^.mabs^.Execute := FALSE;
			d^.home_done := TRUE;
			d^.state := State.HOME_DONE;
		END_IF
	//////\\
	////\\\\
	//\\\\\\
	State.HOME_OFFSET: // địch chuyển tới vị trí HOME_OFFSET
		d^.mabs^.Position := d^.home_offset_μ;
		d^.mabs^.Velocity := d^.home_forward_μ_per_sec;
		d^.mabs^.Acceleration := d^.mabs^.Velocity / d^.ramp_time_sec;
		d^.mabs^.Deceleration := d^.mabs^.Acceleration;
		d^.mabs^.Jerk := d^.mabs^.Acceleration * d^.jerk_factor; // jerk chỉ có tác dụng khi Velocity ramp type khác Trapezoid
		d^.mabs^.Execute := TRUE;
		StateNext(d^.state);
	92:
		IF d^.mabs^.Done THEN // dịch chuyển xong
			d^.mabs^.Execute := FALSE;
			StateNext(d^.state);
		END_IF
	93:
		CASE d^.jog_type OF
			JogType.FSV:
				d^.jog_delta := 0;
				d^.fsv^.dwValueMask := UDINT_TO_DWORD(1 + 2 + 4 + 8);
				d^.fsv^.fSetPosition := d^.home_offset_μ;
				d^.fsv^.fSetVelocity := 0;
				d^.fsv^.fSetAcceleration := 0;
				d^.fsv^.fSetJerk := 0;
				d^.fsv^.bExecute := TRUE;
		END_CASE
		d^.state := State.HOME_OFFSET_DONE;
	//////\\
	////\\\\
	//\\\\\\
	State.READY:
		CASE d^.jog_type OF
			JogType.INCH:
				d^.inch^.Velocity := MIN(d^.max_μ_per_sec, d^.jog_velocity);
				d^.inch^.Acceleration := d^.jog_velocity / d^.ramp_time_sec;
				d^.inch^.Deceleration := d^.inch^.Acceleration;
				d^.inch^.Jerk := d^.inch^.Acceleration * d^.jerk_factor;
				d^.inch^.InchBackward := d^.jog_delta < 0;
				d^.inch^.InchForward := d^.jog_delta > 0;
				IF d^.inch^.InchBackward THEN
					d^.inch^.Distance := d^.ref^.fActPosition;
				END_IF
				IF d^.inch^.InchForward THEN
					d^.inch^.Distance := d^.max_μ - d^.ref^.fActPosition;
				END_IF
			JogType.FSV:
				IF d^.fsv^.bExecute AND NOT d^.fsv^.bError THEN
					d^.fsv^.fSetPosition := MAX(0, MIN(d^.max_μ, d^.fsv^.fSetPosition + d^.jog_delta));
					d^.fsv^.fSetVelocity := MIN(d^.max_μ_per_sec, ABS(d^.jog_velocity));
					d^.fsv^.fSetAcceleration := MIN(d^.max_μ_per_sec * 10, ABS(d^.jog_acceleration));
					d^.fsv^.fSetJerk := d^.fsv^.fSetAcceleration * d^.jerk_factor;
				END_IF
				d^.jog_delta := 0;
		END_CASE
	//////\\
	////\\\\
	//\\\\\\
	State.RUN:
		IF d^.fsv^.bExecute THEN
			d^.fsv^.bExecute := FALSE;
			StateNext(d^.state);
		ELSE
			d^.state := 103;
		END_IF
	102:
		IF NOT d^.fsv^.bError THEN
			StateNext(d^.state);
		END_IF
	103:
		// lệnh chạy đến vị trí chỉ định
		// xem hàm cut() và supply()
		// set d^.target_position_micron và d^.target_velocity_micron_per_sec sau đó set d^.state = State.RUN
		d^.mabs^.Position := MAX(0, MIN(d^.max_μ, d^.target_position_μ)); // giới hạn vị trí, xem save_apply()
		d^.mabs^.Velocity := MAX(0_100, MIN(d^.max_μ_per_sec, d^.target_velocity_μ_per_sec)); // giới hạn tốc độ, xem save_apply()
		d^.mabs^.Acceleration := d^.mabs^.Velocity / d^.ramp_time_sec;
		d^.mabs^.Deceleration := d^.mabs^.Acceleration;
		d^.mabs^.Jerk := d^.mabs^.Acceleration * d^.jerk_factor;
		d^.mabs^.Execute := TRUE;
		StateNext(d^.state);
	104:
		IF d^.mabs^.Done THEN
			d^.mabs^.Execute := FALSE;
			d^.state := State.READY;
		END_IF
END_CASE

ACTION calculate_home_delta_μ:
d^.home_encoder_delta := d^.home_encoder_value_save^ - d^.encoder_single_position;
IF d^.home_encoder_delta >= 0 THEN
	d^.home_delta_μ := ABS(d^.home_encoder_delta) / d^.ref^.fScalefactor;
ELSIF ABS(d^.home_encoder_delta) > (d^.encoder_resolution / 2) THEN
	d^.home_delta_μ := (d^.encoder_resolution - ABS(d^.home_encoder_delta)) / d^.ref^.fScalefactor;
ELSE
	d^.home_delta_μ := -ABS(d^.home_encoder_delta) / d^.ref^.fScalefactor;
END_IF
END_ACTION

METHOD follow
VAR_INPUT
	state: INT;
	follow_data: POINTER TO AxisECFollow;
END_VAR
CASE state OF
	1: // start follow
		follow_data^.self_begin := d^.ref^.fActPosition;
		follow_data^.target_begin := follow_data^.target^.fActPosition;
		follow_data^.offset := 0;
		follow_data^.deviation := 0;
		d^.fsv^.dwValueMask := UDINT_TO_DWORD(1 + 2 + 4 + 8);
		d^.fsv^.fSetPosition := follow_data^.self_begin;
		d^.fsv^.fSetVelocity := 0;
		d^.fsv^.fSetAcceleration := 0;
		d^.fsv^.fSetJerk := 0;
		d^.fsv^.bExecute := TRUE;
	2: // follow
		follow_data^.target_delta := follow_data^.target^.fActPosition - follow_data^.target_begin;
		d^.fsv^.fSetPosition := (follow_data^.self_begin - follow_data^.offset) + (follow_data^.target_delta / follow_data^.ratio);
		d^.fsv^.fSetVelocity := follow_data^.target^.fActVelocity / follow_data^.ratio;
		d^.fsv^.fSetAcceleration := follow_data^.target^.fActAcceleration / follow_data^.ratio;
		d^.fsv^.fSetJerk := follow_data^.target^.fActJerk / follow_data^.ratio;
		follow_data^.deviation := follow_data^.target_delta - (d^.ref^.fActPosition - follow_data^.self_begin + follow_data^.offset) * follow_data^.ratio;
END_CASE
END_METHOD

END_FUNCTION_BLOCK

// Device/Application/AxisFBSetTorqueLimit
FUNCTION_BLOCK AxisFBSetTorqueLimit
VAR_INPUT
	scale_factor: LREAL;
	write: POINTER TO SMC3_ETC_WriteParameter_CoE;
	torque_rated_Nm: LREAL;
	negative_Nm: LREAL;
	positive_Nm: LREAL;
	execute: BOOL;
END_VAR
VAR_OUTPUT
	execute_rise: R_TRIG;
	state: INT;
	done: BOOL;
END_VAR

execute_rise(CLK:= execute, Q=> );
IF execute_rise.Q THEN
	state := 1;
END_IF
IF execute THEN
	CASE state OF
		1:
			done := FALSE;
			IF scale_factor > 0 THEN
				write^.uiIndex := 16#60E1; // servo negative torque limit
			ELSE
				write^.uiIndex := 16#60E0; // servo positive torque limit
			END_IF
			write^.usiSubIndex := 0;
			write^.usiDataLength := 2;
			write^.dwValue := LREAL_TO_DWORD(1000 * (negative_Nm / torque_rated_Nm));
			write^.xExecute := TRUE;
			StateNext(state);
		2:
			IF write^.xDone THEN
				write^.xExecute := FALSE;
				StateNext(state);
			END_IF
		3:
			IF scale_factor > 0 THEN
				write^.uiIndex := 16#60E0; // servo positive torque limit
			ELSE
				write^.uiIndex := 16#60E1; // servo negative torque limit
			END_IF
			write^.usiSubIndex := 0;
			write^.usiDataLength := 2;
			write^.dwValue := LREAL_TO_DWORD(1000 * (positive_Nm / torque_rated_Nm));
			write^.xExecute := TRUE;
			StateNext(state);
		4:
			IF write^.xDone THEN
				write^.xExecute := FALSE;
				done := TRUE;
				state := 0;
			END_IF
	END_CASE
END_IF

END_FUNCTION_BLOCK

// Device/Application/SimpleMotion
FUNCTION_BLOCK SimpleMotion
VAR_INPUT
	state: INT;
	tp: LREAL;
	tv: LREAL;
	ta: LREAL;
	jerk_factor: LREAL;
	dt_sec: LREAL;
END_VAR
VAR_OUTPUT
	p: LREAL;
	v: LREAL;
	a: LREAL;
	d: LREAL;
END_VAR

CASE state OF
	1:
		a := 0;
		v := 0;
		p := 0;
		d := 1;
	2:
		a := MIN(a + d * ta * jerk_factor * dt_sec, ta);
		v := MIN(v + d * a * dt_sec, tv);
		p := MIN(p + v * dt_sec, tp);
		IF p > 0.55 * tp THEN
			d := -1;
		END_IF
END_CASE

END_FUNCTION_BLOCK

// Device/Application/Visualization
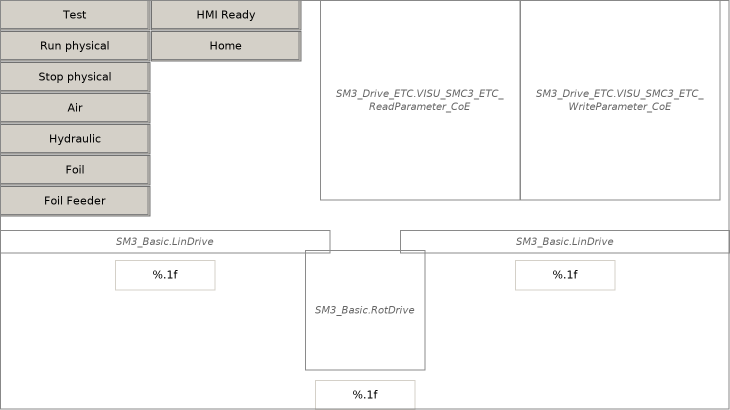
VISUALIZATION Visualization  // 730x410
    Button (0,31 150x30), "Run physical"
        toggle M.work_data.input_run.rise_physical.CLK
    Frame (305,250 120x120)
        shows SM3_Basic.RotDrive(m_Input_AXISREF := M.axiss[2]^)
    Frame (0,230 330x23)
        shows SM3_Basic.LinDrive(m_Input_AXISREF := M.axiss[0]^)
    Frame (400,230 330x23)
        shows SM3_Basic.LinDrive(m_Input_AXISREF := M.axiss[1]^)
    Button (0,0 150x30), "Test"
        toggle M.test
    Button (0,62 150x30), "Stop physical"
        toggle M.work_data.input_stop.fall_physical.CLK
    Button (0,93 150x30), "Air"
        toggle M.supply_data.input_air
    Button (0,124 150x30), "Hydraulic"
        toggle M.supply_data.input_hydraulic
    Button (151,0 150x30), "HMI Ready"
        toggle M.hmi.hmi_ready
    Button (151,31 150x30), "Home"
        toggle M.hmi.home
    Textfield (115,260 100x30), "%.1f", text variable: M.cut_data.axiss[0].home_delta_μ
    Textfield (515,260 100x30), "%.1f", text variable: M.cut_data.axiss[1].home_delta_μ
    Textfield (315,380 100x30), "%.1f", text variable: M.supply_data.axis.home_delta_μ
    Button (0,155 150x30), "Foil"
        toggle M.supply_data.input_foil
    Frame (320,0 200x200)
        shows SM3_Drive_ETC.VISU_SMC3_ETC_ReadParameter_CoE(m_Input_FB := M.axiss_read[0])
    Frame (520,0 200x200)
        shows SM3_Drive_ETC.VISU_SMC3_ETC_WriteParameter_CoE(m_Input_FB := M.axiss_write[0])
    Button (0,186 150x30), "Foil Feeder"
        toggle M.supply_data.input_foil_feeder
END_VISUALIZATION
